LIN {X 0,Y 284.556,Z 208.031,A -85,B 0,C 180,E1 -16929.956,E2 -16929.956} C_VEL
LIN {X 0,Y 284.452,Z 208.046,A -85,B 0,C 180,E1 -16934.304,E2 -16934.304} C_VEL
LIN {X 0,Y 284.322,Z 208.068,A -85,B 0,C 180,E1 -16938.744,E2 -16938.744} C_VEL
LIN {X 0,Y 284.299,Z 208.074,A -85,B 0,C 180,E1 -16943.299,E2 -16943.299} C_VEL
LIN {X 0,Y 284.315,Z 208.073,A -85,B 0,C 180,E1 -16947.146,E2 -16947.146} C_VEL
LIN {X 0,Y 284.286,Z 208.075,A -85,B 0,C 180,E1 -16950.093,E2 -16950.093} C_VEL
LIN {X 0,Y 284.295,Z 208.073,A -85,B 0,C 180,E1 -16952.947,E2 -16952.947} C_VEL
LIN {X 0,Y 284.312,Z 208.07,A -85,B 0,C 180,E1 -16956.389,E2 -16956.389} C_VEL
LIN {X 0,Y 284.299,Z 208.15,A -85,B 0,C 180,E1 -16959.192,E2 -16959.192} C_VEL
LIN {X 0,Y 286.105,Z 215.668,A -85,B 0,C 180,E1 -16963.457,E2 -16963.457} C_VEL
LIN {X 0,Y 287.767,Z 222.743,A -85,B 0,C 180,E1 -16967.111,E2 -16967.111} C_VEL
LIN {X 0,Y 289.38,Z 229.741,A -85,B 0,C 180,E1 -16970.407,E2 -16970.407} C_VEL
LIN {X 0,Y 291.264,Z 238.5,A -85,B 0,C 180,E1 -16974.224,E2 -16974.224} C_VEL
LIN {X 0,Y 292.271,Z 243.914,A -85,B 0,C 180,E1 -16976.425,E2 -16976.425} C_VEL
LIN {X 0,Y 290.199,Z 252.267,A -85,B 0,C 180,E1 -16979.433,E2 -16979.433} C_VEL
LIN {X 0,Y 286.998,Z 266.482,A -85,B 0,C 180,E1 -16984.573,E2 -16984.573} C_VEL
LIN {X 0,Y 285.727,Z 273,A -85,B 0,C 180,E1 -16986.97,E2 -16986.97} C_VEL
LIN {X 0,Y 286.996,Z 286.111,A -85,B 0,C 180,E1 -16987.696,E2 -16987.696} C_VEL
LIN {X 0,Y 287.368,Z 299.101,A -85,B 0,C 180,E1 -16988.692,E2 -16988.692} C_VEL
LIN {X 0,Y 287.659,Z 310.186,A -85,B 0,C 180,E1 -16989.821,E2 -16989.821} C_VEL
LIN {X 0,Y 287.568,Z 320.328,A -85,B 0,C 180,E1 -16991.108,E2 -16991.108} C_VEL
LIN {X 0,Y 286.441,Z 329.749,A -85,B 0,C 180,E1 -16992.511,E2 -16992.511} C_VEL
LIN {X 0,Y 285.855,Z 335.833,A -85,B 0,C 180,E1 -16993.507,E2 -16993.507} C_VEL
LIN {X 0,Y 284.785,Z 346.52,A -85,B 0,C 180,E1 -16995.167,E2 -16995.167} C_VEL
LIN {X 0,Y 283.948,Z 356.755,A -85,B 0,C 180,E1 -16997.131,E2 -16997.131} C_VEL
LIN {X 0,Y 283.401,Z 364.415,A -85,B 0,C 180,E1 -16998.921,E2 -16998.921} C_VEL
LIN {X 0,Y 283.048,Z 371.92,A -85,B 0,C 180,E1 -17001.074,E2 -17001.074} C_VEL
LIN {X 0,Y 282.887,Z 378.816,A -85,B 0,C 180,E1 -17003.595,E2 -17003.595} C_VEL
LIN {X 0,Y 282.821,Z 383.257,A -85,B 0,C 180,E1 -17005.727,E2 -17005.727} C_VEL
LIN {X 0,Y 282.938,Z 385.581,A -85,B 0,C 180,E1 -17007.154,E2 -17007.154} C_VEL
LIN {X 0,Y 282.983,Z 387.424,A -85,B 0,C 180,E1 -17008.579,E2 -17008.579} C_VEL
LIN {X 0,Y 282.977,Z 388.816,A -85,B 0,C 180,E1 -17010.002,E2 -17010.002} C_VEL
LIN {X 0,Y 282.898,Z 389.732,A -85,B 0,C 180,E1 -17011.425,E2 -17011.425} C_VEL
LIN {X 0,Y 282.576,Z 390.303,A -85,B 0,C 180,E1 -17014.281,E2 -17014.281} C_VEL
LIN {X 0,Y 282.524,Z 389.999,A -85,B 0,C 180,E1 -17015.712,E2 -17015.712} C_VEL
LIN {X 0,Y 282.839,Z 388.158,A -85,B 0,C 180,E1 -17018.576,E2 -17018.576} C_VEL
LIN {X 0,Y 283.775,Z 384.776,A -85,B 0,C 180,E1 -17021.429,E2 -17021.429} C_VEL
LIN {X 0,Y 284.906,Z 381.163,A -85,B 0,C 180,E1 -17023.555,E2 -17023.555} C_VEL
LIN {X 0,Y 286.668,Z 376.58,A -85,B 0,C 180,E1 -17025.647,E2 -17025.647} C_VEL
LIN {X 0,Y 288.918,Z 369.965,A -85,B 0,C 180,E1 -17028.07,E2 -17028.07} C_VEL
LIN {X 0,Y 291.48,Z 363.007,A -85,B 0,C 180,E1 -17030.097,E2 -17030.097} C_VEL
LIN {X 0,Y 295.275,Z 353.149,A -85,B 0,C 180,E1 -17032.386,E2 -17032.386} C_VEL
LIN {X 0,Y 298.964,Z 342.899,A -85,B 0,C 180,E1 -17034.294,E2 -17034.294} C_VEL
LIN {X 0,Y 302.662,Z 331.714,A -85,B 0,C 180,E1 -17035.996,E2 -17035.996} C_VEL
LIN {X 0,Y 305.228,Z 321.28,A -85,B 0,C 180,E1 -17037.421,E2 -17037.421} C_VEL
LIN {X 0,Y 306.812,Z 309.853,A -85,B 0,C 180,E1 -17038.948,E2 -17038.948} C_VEL
LIN {X 0,Y 307.335,Z 299.297,A -85,B 0,C 180,E1 -17040.382,E2 -17040.382} C_VEL
LIN {X 0,Y 306.766,Z 286.625,A -85,B 0,C 180,E1 -17042.257,E2 -17042.257} C_VEL
LIN {X 0,Y 305.752,Z 277.475,A -85,B 0,C 180,E1 -17043.754,E2 -17043.754} C_VEL
LIN {X 0,Y 304.821,Z 269.242,A -85,B 0,C 180,E1 -17045.302,E2 -17045.302} C_VEL
LIN {X 0,Y 305.142,Z 266.775,A -85,B 0,C 180,E1 -17046.281,E2 -17046.281} C_VEL
LIN {X 0,Y 305.029,Z 262.987,A -85,B 0,C 180,E1 -17048.471,E2 -17048.471} C_VEL
LIN {X 0,Y 304.799,Z 260.629,A -85,B 0,C 180,E1 -17050.456,E2 -17050.456} C_VEL
LIN {X 0,Y 304.213,Z 259.405,A -85,B 0,C 180,E1 -17052.33,E2 -17052.33} C_VEL
LIN {X 0,Y 303.415,Z 259.011,A -85,B 0,C 180,E1 -17054.106,E2 -17054.106} C_VEL
LIN {X 0,Y 302.635,Z 259.068,A -85,B 0,C 180,E1 -17056.048,E2 -17056.048} C_VEL
LIN {X 0,Y 301.48,Z 260.13,A -85,B 0,C 180,E1 -17059.252,E2 -17059.252} C_VEL
LIN {X 0,Y 300.921,Z 261.159,A -85,B 0,C 180,E1 -17060.907,E2 -17060.907} C_VEL
LIN {X 0,Y 300.012,Z 262.974,A -85,B 0,C 180,E1 -17062.651,E2 -17062.651} C_VEL
LIN {X 0,Y 301.617,Z 268.449,A -85,B 0,C 180,E1 -17064.643,E2 -17064.643} C_VEL
LIN {X 0,Y 304.148,Z 276.846,A -85,B 0,C 180,E1 -17067.224,E2 -17067.224} C_VEL
LIN {X 0,Y 306.842,Z 287.914,A -85,B 0,C 180,E1 -17070.05,E2 -17070.05} C_VEL
LIN {X 0,Y 308.147,Z 297.139,A -85,B 0,C 180,E1 -17072.074,E2 -17072.074} C_VEL
LIN {X 0,Y 308.384,Z 304.136,A -85,B 0,C 180,E1 -17073.478,E2 -17073.478} C_VEL
LIN {X 0,Y 304.667,Z 315.586,A -85,B 0,C 180,E1 -17075.103,E2 -17075.103} C_VEL
LIN {X 0,Y 300.868,Z 326.03,A -85,B 0,C 180,E1 -17076.967,E2 -17076.967} C_VEL
LIN {X 0,Y 297.408,Z 334.701,A -85,B 0,C 180,E1 -17078.877,E2 -17078.877} C_VEL
LIN {X 0,Y 293.88,Z 342.88,A -85,B 0,C 180,E1 -17081.165,E2 -17081.165} C_VEL
LIN {X 0,Y 291.288,Z 348.565,A -85,B 0,C 180,E1 -17083.17,E2 -17083.17} C_VEL
LIN {X 0,Y 289.185,Z 353.139,A -85,B 0,C 180,E1 -17085.216,E2 -17085.216} C_VEL
LIN {X 0,Y 287.297,Z 356.739,A -85,B 0,C 180,E1 -17087.281,E2 -17087.281} C_VEL
LIN {X 0,Y 285.522,Z 359.952,A -85,B 0,C 180,E1 -17089.933,E2 -17089.933} C_VEL
LIN {X 0,Y 284.505,Z 361.163,A -85,B 0,C 180,E1 -17091.477,E2 -17091.477} C_VEL
LIN {X 0,Y 283.599,Z 362.166,A -85,B 0,C 180,E1 -17094.311,E2 -17094.311} C_VEL
LIN {X 0,Y 283.258,Z 362.063,A -85,B 0,C 180,E1 -17095.731,E2 -17095.731} C_VEL
LIN {X 0,Y 282.702,Z 360.712,A -85,B 0,C 180,E1 -17098.576,E2 -17098.576} C_VEL
LIN {X 0,Y 282.565,Z 359.447,A -85,B 0,C 180,E1 -17100,E2 -17100} C_VEL
LIN {X 0,Y 282.563,Z 356.745,A -85,B 0,C 180,E1 -17102.138,E2 -17102.138} C_VEL
LIN {X 0,Y 282.716,Z 353.044,A -85,B 0,C 180,E1 -17104.277,E2 -17104.277} C_VEL
LIN {X 0,Y 282.917,Z 347.475,A -85,B 0,C 180,E1 -17106.712,E2 -17106.712} C_VEL
LIN {X 0,Y 283.339,Z 341.061,A -85,B 0,C 180,E1 -17108.918,E2 -17108.918} C_VEL
LIN {X 0,Y 283.988,Z 333.386,A -85,B 0,C 180,E1 -17111.058,E2 -17111.058} C_VEL
LIN {X 0,Y 284.831,Z 323.888,A -85,B 0,C 180,E1 -17113.193,E2 -17113.193} C_VEL
LIN {X 0,Y 285.828,Z 314.315,A -85,B 0,C 180,E1 -17114.962,E2 -17114.962} C_VEL
LIN {X 0,Y 286.847,Z 302.522,A -85,B 0,C 180,E1 -17116.732,E2 -17116.732} C_VEL
LIN {X 0,Y 287.821,Z 291.265,A -85,B 0,C 180,E1 -17118.103,E2 -17118.103} C_VEL
LIN {X 0,Y 288.584,Z 280.158,A -85,B 0,C 180,E1 -17119.194,E2 -17119.194} C_VEL
LIN {X 0,Y 286.473,Z 266.68,A -85,B 0,C 180,E1 -17120.318,E2 -17120.318} C_VEL
LIN {X 0,Y 284.567,Z 252.884,A -85,B 0,C 180,E1 -17121.173,E2 -17121.173} C_VEL
LIN {X 0,Y 284.521,Z 252.298,A -85,B 0,C 180,E1 -17121.24,E2 -17121.24} C_VEL
LIN {X 0,Y 284.94,Z 244.617,A -85,B 0,C 180,E1 -17124.791,E2 -17124.791} C_VEL
LIN {X 0,Y 285.368,Z 236.232,A -85,B 0,C 180,E1 -17128.702,E2 -17128.702} C_VEL
LIN {X 0,Y 285.937,Z 227.639,A -85,B 0,C 180,E1 -17132.734,E2 -17132.734} C_VEL
LIN {X 0,Y 286.29,Z 220.567,A -85,B 0,C 180,E1 -17136.098,E2 -17136.098} C_VEL
LIN {X 0,Y 285.648,Z 214.901,A -85,B 0,C 180,E1 -17138.886,E2 -17138.886} C_VEL
LIN {X 0,Y 284.363,Z 208.065,A -85,B 0,C 180,E1 -17142.352,E2 -17142.352} C_VEL
LIN {X 0,Y 284.262,Z 208.078,A -85,B 0,C 180,E1 -17146.188,E2 -17146.188} C_VEL
LIN {X 0,Y 284.312,Z 208.072,A -85,B 0,C 180,E1 -17150.023,E2 -17150.023} C_VEL
LIN {X 0,Y 284.326,Z 208.072,A -85,B 0,C 180,E1 -17153.611,E2 -17153.611} C_VEL
LIN {X 0,Y 284.368,Z 208.282,A -85,B 0,C 180,E1 -17155.007,E2 -17155.007} C_VEL
LIN {X 0,Y 284.692,Z 210.194,A -85,B 0,C 180,E1 -17157.103,E2 -17157.103} C_VEL
LIN {X 0,Y 284.913,Z 213.447,A -85,B 0,C 180,E1 -17160.438,E2 -17160.438} C_VEL
LIN {X 0,Y 284.838,Z 216.778,A -85,B 0,C 180,E1 -17163.631,E2 -17163.631} C_VEL
LIN {X 0,Y 284.709,Z 220.161,A -85,B 0,C 180,E1 -17166.735,E2 -17166.735} C_VEL
LIN {X 0,Y 284.654,Z 223.645,A -85,B 0,C 180,E1 -17169.776,E2 -17169.776} C_VEL
LIN {X 0,Y 284.578,Z 226.72,A -85,B 0,C 180,E1 -17172.321,E2 -17172.321} C_VEL
LIN {X 0,Y 287.73,Z 237.495,A -85,B 0,C 180,E1 -17173.172,E2 -17173.172} C_VEL
LIN {X 0,Y 290.174,Z 247.752,A -85,B 0,C 180,E1 -17174.248,E2 -17174.248} C_VEL
LIN {X 0,Y 291.01,Z 253.902,A -85,B 0,C 180,E1 -17175.021,E2 -17175.021} C_VEL
LIN {X 0,Y 290.089,Z 263.238,A -85,B 0,C 180,E1 -17176.335,E2 -17176.335} C_VEL
LIN {X 0,Y 289.359,Z 269.037,A -85,B 0,C 180,E1 -17177.372,E2 -17177.372} C_VEL
LIN {X 0,Y 288.305,Z 275.346,A -85,B 0,C 180,E1 -17178.753,E2 -17178.753} C_VEL
LIN {X 0,Y 287.394,Z 280.335,A -85,B 0,C 180,E1 -17180.142,E2 -17180.142} C_VEL
LIN {X 0,Y 286.592,Z 284.326,A -85,B 0,C 180,E1 -17181.537,E2 -17181.537} C_VEL
LIN {X 0,Y 286.092,Z 288.746,A -85,B 0,C 180,E1 -17183.652,E2 -17183.652} C_VEL
LIN {X 0,Y 285.241,Z 291.75,A -85,B 0,C 180,E1 -17185.759,E2 -17185.759} C_VEL
LIN {X 0,Y 285.065,Z 293.009,A -85,B 0,C 180,E1 -17187.172,E2 -17187.172} C_VEL
LIN {X 0,Y 284.86,Z 293.775,A -85,B 0,C 180,E1 -17188.584,E2 -17188.584} C_VEL
LIN {X 0,Y 284.777,Z 294.043,A -85,B 0,C 180,E1 -17189.998,E2 -17189.998} C_VEL
LIN {X 0,Y 284.858,Z 293.811,A -85,B 0,C 180,E1 -17191.412,E2 -17191.412} C_VEL
LIN {X 0,Y 285.061,Z 293.095,A -85,B 0,C 180,E1 -17192.824,E2 -17192.824} C_VEL
LIN {X 0,Y 285.238,Z 291.887,A -85,B 0,C 180,E1 -17194.237,E2 -17194.237} C_VEL
LIN {X 0,Y 286.082,Z 288.958,A -85,B 0,C 180,E1 -17196.345,E2 -17196.345} C_VEL
LIN {X 0,Y 286.554,Z 284.623,A -85,B 0,C 180,E1 -17198.46,E2 -17198.46} C_VEL
LIN {X 0,Y 287.252,Z 281.745,A -85,B 0,C 180,E1 -17199.504,E2 -17199.504} C_VEL
LIN {X 0,Y 288.046,Z 277.103,A -85,B 0,C 180,E1 -17200.898,E2 -17200.898} C_VEL
LIN {X 0,Y 289.079,Z 271.275,A -85,B 0,C 180,E1 -17202.28,E2 -17202.28} C_VEL
LIN {X 0,Y 289.917,Z 264.953,A -85,B 0,C 180,E1 -17203.491,E2 -17203.491} C_VEL
LIN {X 0,Y 290.611,Z 257.713,A -85,B 0,C 180,E1 -17204.606,E2 -17204.606} C_VEL
LIN {X 0,Y 291.046,Z 252.834,A -85,B 0,C 180,E1 -17205.231,E2 -17205.231} C_VEL
LIN {X 0,Y 289.66,Z 245.069,A -85,B 0,C 180,E1 -17206.177,E2 -17206.177} C_VEL
LIN {X 0,Y 286.946,Z 234.411,A -85,B 0,C 180,E1 -17207.213,E2 -17207.213} C_VEL
LIN {X 0,Y 284.582,Z 226.689,A -85,B 0,C 180,E1 -17207.839,E2 -17207.839} C_VEL
LIN {X 0,Y 284.672,Z 223.765,A -85,B 0,C 180,E1 -17210.256,E2 -17210.256} C_VEL
LIN {X 0,Y 284.791,Z 218.619,A -85,B 0,C 180,E1 -17214.802,E2 -17214.802} C_VEL
LIN {X 0,Y 284.886,Z 215.255,A -85,B 0,C 180,E1 -17217.949,E2 -17217.949} C_VEL
LIN {X 0,Y 284.815,Z 211.982,A -85,B 0,C 180,E1 -17221.208,E2 -17221.208} C_VEL
LIN {X 0,Y 284.444,Z 208.769,A -85,B 0,C 180,E1 -17224.628,E2 -17224.628} C_VEL
LIN {X 0,Y 284.344,Z 208.067,A -85,B 0,C 180,E1 -17225.512,E2 -17225.512} C_VEL
LIN {X 0,Y 284.318,Z 208.069,A -85,B 0,C 180,E1 -17228.165,E2 -17228.165} C_VEL
LIN {X 0,Y 284.263,Z 208.075,A -85,B 0,C 180,E1 -17232.123,E2 -17232.123} C_VEL
LIN {X 0,Y 284.279,Z 208.071,A -85,B 0,C 180,E1 -17236.193,E2 -17236.193} C_VEL
LIN {X 0,Y 284.305,Z 208.067,A -85,B 0,C 180,E1 -17240.021,E2 -17240.021} C_VEL
LIN {X 0,Y 284.326,Z 208.066,A -85,B 0,C 180,E1 -17243.613,E2 -17243.613} C_VEL
LIN {X 0,Y 284.301,Z 208.067,A -85,B 0,C 180,E1 -17247.188,E2 -17247.188} C_VEL
LIN {X 0,Y 284.351,Z 208.056,A -85,B 0,C 180,E1 -17250.375,E2 -17250.375} C_VEL
LIN {X 0,Y 284.369,Z 208.061,A -85,B 0,C 180,E1 -17253.585,E2 -17253.585} C_VEL
LIN {X 0,Y 284.357,Z 208.064,A -85,B 0,C 180,E1 -17256.706,E2 -17256.706} C_VEL
LIN {X 0,Y 284.394,Z 208.056,A -85,B 0,C 180,E1 -17261.261,E2 -17261.261} C_VEL
LIN {X 0,Y 284.482,Z 208.035,A -85,B 0,C 180,E1 -17264.458,E2 -17264.458} C_VEL
LIN {X 0,Y 284.477,Z 208.046,A -85,B 0,C 180,E1 -17268.601,E2 -17268.601} C_VEL
LIN {X 0,Y 284.628,Z 208.024,A -85,B 0,C 180,E1 -17271.48,E2 -17271.48} C_VEL
LIN {X 0,Y 284.586,Z 208.026,A -85,B 0,C 180,E1 -17274.331,E2 -17274.331} C_VEL
LIN {X 0,Y 284.844,Z 207.997,A -85,B 0,C 180,E1 -17278.76,E2 -17278.76} C_VEL
LIN {X 0,Y 284.138,Z 208.08,A -85,B 0,C 180,E1 -17279.941,E2 -17279.941} C_VEL
LIN {X 0,Y 281.114,Z 208.466,A -85,B 0,C 180,E1 -17281.859,E2 -17281.859} C_VEL
LIN {X 0,Y 278.579,Z 208.78,A -85,B 0,C 180,E1 -17283.418,E2 -17283.418} C_VEL
LIN {X 0,Y 277.537,Z 208.903,A -85,B 0,C 180,E1 -17284.63,E2 -17284.63} C_VEL
LIN {X 0,Y 277.478,Z 208.911,A -85,B 0,C 180,E1 -17285.041,E2 -17285.041} C_VEL
LIN {X 0,Y 277.642,Z 208.9,A -85,B 0,C 180,E1 -17287.271,E2 -17287.271} C_VEL
LIN {X 0,Y 277.496,Z 208.912,A -85,B 0,C 180,E1 -17290.212,E2 -17290.212} C_VEL
LIN {X 0,Y 277.398,Z 208.928,A -85,B 0,C 180,E1 -17294.676,E2 -17294.676} C_VEL
LIN {X 0,Y 277.274,Z 208.948,A -85,B 0,C 180,E1 -17299.239,E2 -17299.239} C_VEL
LIN {X 0,Y 277.249,Z 208.952,A -85,B 0,C 180,E1 -17303.928,E2 -17303.928} C_VEL
LIN {X 0,Y 277.256,Z 208.951,A -85,B 0,C 180,E1 -17307.482,E2 -17307.482} C_VEL
LIN {X 0,Y 277.238,Z 208.952,A -85,B 0,C 180,E1 -17310.474,E2 -17310.474} C_VEL
LIN {X 0,Y 277.236,Z 208.947,A -85,B 0,C 180,E1 -17313.897,E2 -17313.897} C_VEL
LIN {X 0,Y 277.263,Z 208.948,A -85,B 0,C 180,E1 -17317.845,E2 -17317.845} C_VEL
LIN {X 0,Y 277.289,Z 209.153,A -85,B 0,C 180,E1 -17318.218,E2 -17318.218} C_VEL
LIN {X 0,Y 278.743,Z 215.264,A -85,B 0,C 180,E1 -17321.925,E2 -17321.925} C_VEL
LIN {X 0,Y 280.48,Z 222.527,A -85,B 0,C 180,E1 -17325.832,E2 -17325.832} C_VEL
LIN {X 0,Y 282.263,Z 230.179,A -85,B 0,C 180,E1 -17329.659,E2 -17329.659} C_VEL
LIN {X 0,Y 284.092,Z 238.844,A -85,B 0,C 180,E1 -17333.581,E2 -17333.581} C_VEL
LIN {X 0,Y 285.287,Z 245.368,A -85,B 0,C 180,E1 -17336.342,E2 -17336.342} C_VEL
LIN {X 0,Y 282.547,Z 255.692,A -85,B 0,C 180,E1 -17340.169,E2 -17340.169} C_VEL
LIN {X 0,Y 279.795,Z 267.845,A -85,B 0,C 180,E1 -17344.724,E2 -17344.724} C_VEL
LIN {X 0,Y 278.89,Z 272.292,A -85,B 0,C 180,E1 -17346.421,E2 -17346.421} C_VEL
LIN {X 0,Y 280.198,Z 286.506,A -85,B 0,C 180,E1 -17347.27,E2 -17347.27} C_VEL
LIN {X 0,Y 280.535,Z 297.591,A -85,B 0,C 180,E1 -17348.147,E2 -17348.147} C_VEL
LIN {X 0,Y 280.705,Z 309.027,A -85,B 0,C 180,E1 -17349.319,E2 -17349.319} C_VEL
LIN {X 0,Y 280.696,Z 319.136,A -85,B 0,C 180,E1 -17350.627,E2 -17350.627} C_VEL
LIN {X 0,Y 279.807,Z 327.565,A -85,B 0,C 180,E1 -17351.893,E2 -17351.893} C_VEL
LIN {X 0,Y 278.362,Z 339.738,A -85,B 0,C 180,E1 -17354.066,E2 -17354.066} C_VEL
LIN {X 0,Y 277.479,Z 349.307,A -85,B 0,C 180,E1 -17355.705,E2 -17355.705} C_VEL
LIN {X 0,Y 276.636,Z 359.657,A -85,B 0,C 180,E1 -17357.904,E2 -17357.904} C_VEL
LIN {X 0,Y 276.09,Z 368.004,A -85,B 0,C 180,E1 -17360.108,E2 -17360.108} C_VEL
LIN {X 0,Y 275.934,Z 373.705,A -85,B 0,C 180,E1 -17361.949,E2 -17361.949} C_VEL
LIN {X 0,Y 275.856,Z 379.204,A -85,B 0,C 180,E1 -17364.153,E2 -17364.153} C_VEL
LIN {X 0,Y 275.829,Z 383.434,A -85,B 0,C 180,E1 -17366.35,E2 -17366.35} C_VEL
LIN {X 0,Y 275.93,Z 386.546,A -85,B 0,C 180,E1 -17368.542,E2 -17368.542} C_VEL
LIN {X 0,Y 275.922,Z 388.02,A -85,B 0,C 180,E1 -17370.002,E2 -17370.002} C_VEL
LIN {X 0,Y 275.833,Z 389.057,A -85,B 0,C 180,E1 -17371.462,E2 -17371.462} C_VEL
LIN {X 0,Y 275.515,Z 389.644,A -85,B 0,C 180,E1 -17372.926,E2 -17372.926} C_VEL
LIN {X 0,Y 275.453,Z 389.649,A -85,B 0,C 180,E1 -17375.696,E2 -17375.696} C_VEL
LIN {X 0,Y 275.526,Z 389.004,A -85,B 0,C 180,E1 -17377.329,E2 -17377.329} C_VEL
LIN {X 0,Y 275.797,Z 388.026,A -85,B 0,C 180,E1 -17378.797,E2 -17378.797} C_VEL
LIN {X 0,Y 276.795,Z 384.854,A -85,B 0,C 180,E1 -17381.722,E2 -17381.722} C_VEL
LIN {X 0,Y 277.992,Z 381.459,A -85,B 0,C 180,E1 -17383.898,E2 -17383.898} C_VEL
LIN {X 0,Y 280.551,Z 375.462,A -85,B 0,C 180,E1 -17386.745,E2 -17386.745} C_VEL
LIN {X 0,Y 283.08,Z 368.624,A -85,B 0,C 180,E1 -17389.244,E2 -17389.244} C_VEL
LIN {X 0,Y 286.534,Z 360.394,A -85,B 0,C 180,E1 -17391.589,E2 -17391.589} C_VEL
LIN {X 0,Y 290.099,Z 351.783,A -85,B 0,C 180,E1 -17393.563,E2 -17393.563} C_VEL
LIN {X 0,Y 294.129,Z 341.451,A -85,B 0,C 180,E1 -17395.475,E2 -17395.475} C_VEL
LIN {X 0,Y 297.935,Z 330.338,A -85,B 0,C 180,E1 -17397.198,E2 -17397.198} C_VEL
LIN {X 0,Y 300.617,Z 319.331,A -85,B 0,C 180,E1 -17398.76,E2 -17398.76} C_VEL
LIN {X 0,Y 302.234,Z 307.982,A -85,B 0,C 180,E1 -17400.358,E2 -17400.358} C_VEL
LIN {X 0,Y 302.693,Z 296.454,A -85,B 0,C 180,E1 -17402.099,E2 -17402.099} C_VEL
LIN {X 0,Y 302.356,Z 285.308,A -85,B 0,C 180,E1 -17403.91,E2 -17403.91} C_VEL
LIN {X 0,Y 301.381,Z 274.903,A -85,B 0,C 180,E1 -17405.87,E2 -17405.87} C_VEL
LIN {X 0,Y 300.858,Z 272.433,A -85,B 0,C 180,E1 -17406.511,E2 -17406.511} C_VEL
LIN {X 0,Y 299.528,Z 268.255,A -85,B 0,C 180,E1 -17408.065,E2 -17408.065} C_VEL
LIN {X 0,Y 299.467,Z 266.402,A -85,B 0,C 180,E1 -17409.321,E2 -17409.321} C_VEL
LIN {X 0,Y 299.006,Z 264.514,A -85,B 0,C 180,E1 -17411.223,E2 -17411.223} C_VEL
LIN {X 0,Y 298.23,Z 263.565,A -85,B 0,C 180,E1 -17413.112,E2 -17413.112} C_VEL
LIN {X 0,Y 297.267,Z 263.279,A -85,B 0,C 180,E1 -17415.177,E2 -17415.177} C_VEL
LIN {X 0,Y 295.998,Z 263.852,A -85,B 0,C 180,E1 -17418.332,E2 -17418.332} C_VEL
LIN {X 0,Y 295.723,Z 264.277,A -85,B 0,C 180,E1 -17419.189,E2 -17419.189} C_VEL
LIN {X 0,Y 297.195,Z 268.792,A -85,B 0,C 180,E1 -17422.059,E2 -17422.059} C_VEL
LIN {X 0,Y 298.351,Z 273.545,A -85,B 0,C 180,E1 -17423.921,E2 -17423.921} C_VEL
LIN {X 0,Y 300.127,Z 281.201,A -85,B 0,C 180,E1 -17426.42,E2 -17426.42} C_VEL
LIN {X 0,Y 302.144,Z 291.405,A -85,B 0,C 180,E1 -17429.221,E2 -17429.221} C_VEL
LIN {X 0,Y 303.018,Z 299.258,A -85,B 0,C 180,E1 -17431.089,E2 -17431.089} C_VEL
LIN {X 0,Y 303.194,Z 305.086,A -85,B 0,C 180,E1 -17432.38,E2 -17432.38} C_VEL
LIN {X 0,Y 303.03,Z 306.944,A -85,B 0,C 180,E1 -17432.745,E2 -17432.745} C_VEL
LIN {X 0,Y 299.389,Z 317.16,A -85,B 0,C 180,E1 -17434.261,E2 -17434.261} C_VEL
LIN {X 0,Y 295.34,Z 327.36,A -85,B 0,C 180,E1 -17436.138,E2 -17436.138} C_VEL
LIN {X 0,Y 291.691,Z 335.803,A -85,B 0,C 180,E1 -17438.071,E2 -17438.071} C_VEL
LIN {X 0,Y 287.904,Z 343.832,A -85,B 0,C 180,E1 -17440.388,E2 -17440.388} C_VEL
LIN {X 0,Y 284.688,Z 350.235,A -85,B 0,C 180,E1 -17442.768,E2 -17442.768} C_VEL
LIN {X 0,Y 282.463,Z 354.544,A -85,B 0,C 180,E1 -17444.856,E2 -17444.856} C_VEL
LIN {X 0,Y 280.498,Z 357.916,A -85,B 0,C 180,E1 -17446.968,E2 -17446.968} C_VEL
LIN {X 0,Y 278.517,Z 360.953,A -85,B 0,C 180,E1 -17449.826,E2 -17449.826} C_VEL
LIN {X 0,Y 277.528,Z 361.939,A -85,B 0,C 180,E1 -17451.261,E2 -17451.261} C_VEL
LIN {X 0,Y 276.917,Z 362.505,A -85,B 0,C 180,E1 -17452.71,E2 -17452.71} C_VEL
LIN {X 0,Y 276.548,Z 362.662,A -85,B 0,C 180,E1 -17454.166,E2 -17454.166} C_VEL
LIN {X 0,Y 276.191,Z 362.455,A -85,B 0,C 180,E1 -17455.622,E2 -17455.622} C_VEL
LIN {X 0,Y 275.842,Z 361.877,A -85,B 0,C 180,E1 -17457.079,E2 -17457.079} C_VEL
LIN {X 0,Y 275.616,Z 360.891,A -85,B 0,C 180,E1 -17458.539,E2 -17458.539} C_VEL
LIN {X 0,Y 275.466,Z 357.675,A -85,B 0,C 180,E1 -17461.462,E2 -17461.462} C_VEL
LIN {X 0,Y 275.601,Z 354.143,A -85,B 0,C 180,E1 -17463.655,E2 -17463.655} C_VEL
LIN {X 0,Y 275.724,Z 348.651,A -85,B 0,C 180,E1 -17466.224,E2 -17466.224} C_VEL
LIN {X 0,Y 276.218,Z 341.497,A -85,B 0,C 180,E1 -17468.781,E2 -17468.781} C_VEL
LIN {X 0,Y 276.845,Z 333.843,A -85,B 0,C 180,E1 -17470.976,E2 -17470.976} C_VEL
LIN {X 0,Y 277.684,Z 324.356,A -85,B 0,C 180,E1 -17473.167,E2 -17473.167} C_VEL
LIN {X 0,Y 278.794,Z 313.745,A -85,B 0,C 180,E1 -17475.162,E2 -17475.162} C_VEL
LIN {X 0,Y 279.753,Z 303.135,A -85,B 0,C 180,E1 -17476.788,E2 -17476.788} C_VEL
LIN {X 0,Y 280.755,Z 291.635,A -85,B 0,C 180,E1 -17478.234,E2 -17478.234} C_VEL
LIN {X 0,Y 281.534,Z 281.007,A -85,B 0,C 180,E1 -17479.315,E2 -17479.315} C_VEL
LIN {X 0,Y 279.378,Z 266.893,A -85,B 0,C 180,E1 -17480.525,E2 -17480.525} C_VEL
LIN {X 0,Y 277.475,Z 252.691,A -85,B 0,C 180,E1 -17481.439,E2 -17481.439} C_VEL
LIN {X 0,Y 277.966,Z 244.118,A -85,B 0,C 180,E1 -17485.457,E2 -17485.457} C_VEL
LIN {X 0,Y 278.417,Z 235.601,A -85,B 0,C 180,E1 -17489.488,E2 -17489.488} C_VEL
LIN {X 0,Y 278.932,Z 228.638,A -85,B 0,C 180,E1 -17492.801,E2 -17492.801} C_VEL
LIN {X 0,Y 279.27,Z 222.266,A -85,B 0,C 180,E1 -17495.859,E2 -17495.859} C_VEL
LIN {X 0,Y 278.964,Z 218.209,A -85,B 0,C 180,E1 -17497.876,E2 -17497.876} C_VEL
LIN {X 0,Y 277.632,Z 210.663,A -85,B 0,C 180,E1 -17501.687,E2 -17501.687} C_VEL
LIN {X 0,Y 277.304,Z 208.945,A -85,B 0,C 180,E1 -17502.626,E2 -17502.626} C_VEL
LIN {X 0,Y 277.221,Z 208.952,A -85,B 0,C 180,E1 -17507.324,E2 -17507.324} C_VEL
LIN {X 0,Y 277.262,Z 208.953,A -85,B 0,C 180,E1 -17511.794,E2 -17511.794} C_VEL
LIN {X 0,Y 277.305,Z 209.052,A -85,B 0,C 180,E1 -17514.195,E2 -17514.195} C_VEL
LIN {X 0,Y 277.805,Z 212.464,A -85,B 0,C 180,E1 -17517.907,E2 -17517.907} C_VEL
LIN {X 0,Y 277.931,Z 215.745,A -85,B 0,C 180,E1 -17521.283,E2 -17521.283} C_VEL
LIN {X 0,Y 277.823,Z 220.273,A -85,B 0,C 180,E1 -17525.6,E2 -17525.6} C_VEL
LIN {X 0,Y 277.672,Z 224.609,A -85,B 0,C 180,E1 -17529.47,E2 -17529.47} C_VEL
LIN {X 0,Y 277.613,Z 227.461,A -85,B 0,C 180,E1 -17531.793,E2 -17531.793} C_VEL
LIN {X 0,Y 280.661,Z 237.687,A -85,B 0,C 180,E1 -17532.625,E2 -17532.625} C_VEL
LIN {X 0,Y 283.139,Z 247.63,A -85,B 0,C 180,E1 -17533.689,E2 -17533.689} C_VEL
LIN {X 0,Y 284.219,Z 255.206,A -85,B 0,C 180,E1 -17534.66,E2 -17534.66} C_VEL
LIN {X 0,Y 283.283,Z 264.343,A -85,B 0,C 180,E1 -17536,E2 -17536} C_VEL
LIN {X 0,Y 282.522,Z 270.096,A -85,B 0,C 180,E1 -17537.061,E2 -17537.061} C_VEL
LIN {X 0,Y 281.424,Z 276.38,A -85,B 0,C 180,E1 -17538.474,E2 -17538.474} C_VEL
LIN {X 0,Y 280.473,Z 281.342,A -85,B 0,C 180,E1 -17539.896,E2 -17539.896} C_VEL
LIN {X 0,Y 279.641,Z 285.319,A -85,B 0,C 180,E1 -17541.325,E2 -17541.325} C_VEL
LIN {X 0,Y 279.108,Z 289.729,A -85,B 0,C 180,E1 -17543.492,E2 -17543.492} C_VEL
LIN {X 0,Y 278.234,Z 292.727,A -85,B 0,C 180,E1 -17545.652,E2 -17545.652} C_VEL
LIN {X 0,Y 278.046,Z 293.984,A -85,B 0,C 180,E1 -17547.1,E2 -17547.1} C_VEL
LIN {X 0,Y 277.835,Z 294.749,A -85,B 0,C 180,E1 -17548.549,E2 -17548.549} C_VEL
LIN {X 0,Y 277.75,Z 295.017,A -85,B 0,C 180,E1 -17549.998,E2 -17549.998} C_VEL
LIN {X 0,Y 277.833,Z 294.784,A -85,B 0,C 180,E1 -17551.448,E2 -17551.448} C_VEL
LIN {X 0,Y 278.043,Z 294.068,A -85,B 0,C 180,E1 -17552.896,E2 -17552.896} C_VEL
LIN {X 0,Y 278.231,Z 292.862,A -85,B 0,C 180,E1 -17554.344,E2 -17554.344} C_VEL
LIN {X 0,Y 279.098,Z 289.935,A -85,B 0,C 180,E1 -17556.505,E2 -17556.505} C_VEL
LIN {X 0,Y 279.603,Z 285.609,A -85,B 0,C 180,E1 -17558.672,E2 -17558.672} C_VEL
LIN {X 0,Y 280.322,Z 282.745,A -85,B 0,C 180,E1 -17559.741,E2 -17559.741} C_VEL
LIN {X 0,Y 281.148,Z 278.129,A -85,B 0,C 180,E1 -17561.169,E2 -17561.169} C_VEL
LIN {X 0,Y 282.228,Z 272.329,A -85,B 0,C 180,E1 -17562.583,E2 -17562.583} C_VEL
LIN {X 0,Y 283.109,Z 266.05,A -85,B 0,C 180,E1 -17563.822,E2 -17563.822} C_VEL
LIN {X 0,Y 283.832,Z 258.789,A -85,B 0,C 180,E1 -17564.976,E2 -17564.976} C_VEL
LIN {X 0,Y 284.247,Z 254.012,A -85,B 0,C 180,E1 -17565.612,E2 -17565.612} C_VEL
LIN {X 0,Y 282.588,Z 244.937,A -85,B 0,C 180,E1 -17566.745,E2 -17566.745} C_VEL
LIN {X 0,Y 279.806,Z 234.363,A -85,B 0,C 180,E1 -17567.79,E2 -17567.79} C_VEL
LIN {X 0,Y 277.624,Z 227.362,A -85,B 0,C 180,E1 -17568.349,E2 -17568.349} C_VEL
LIN {X 0,Y 277.689,Z 222.743,A -85,B 0,C 180,E1 -17572.309,E2 -17572.309} C_VEL
LIN {X 0,Y 277.823,Z 219.272,A -85,B 0,C 180,E1 -17575.468,E2 -17575.468} C_VEL
LIN {X 0,Y 277.932,Z 215.916,A -85,B 0,C 180,E1 -17578.712,E2 -17578.712} C_VEL
LIN {X 0,Y 277.911,Z 213.917,A -85,B 0,C 180,E1 -17580.704,E2 -17580.704} C_VEL
LIN {X 0,Y 277.589,Z 210.965,A -85,B 0,C 180,E1 -17583.846,E2 -17583.846} C_VEL
LIN {X 0,Y 277.294,Z 208.945,A -85,B 0,C 180,E1 -17586.12,E2 -17586.12} C_VEL
LIN {X 0,Y 277.233,Z 208.952,A -85,B 0,C 180,E1 -17589.325,E2 -17589.325} C_VEL
LIN {X 0,Y 277.21,Z 208.954,A -85,B 0,C 180,E1 -17593.195,E2 -17593.195} C_VEL
LIN {X 0,Y 277.231,Z 208.951,A -85,B 0,C 180,E1 -17597.318,E2 -17597.318} C_VEL
LIN {X 0,Y 277.263,Z 208.946,A -85,B 0,C 180,E1 -17601.789,E2 -17601.789} C_VEL
LIN {X 0,Y 277.277,Z 208.947,A -85,B 0,C 180,E1 -17604.34,E2 -17604.34} C_VEL
LIN {X 0,Y 277.238,Z 208.95,A -85,B 0,C 180,E1 -17607.835,E2 -17607.835} C_VEL
LIN {X 0,Y 277.281,Z 208.939,A -85,B 0,C 180,E1 -17611.211,E2 -17611.211} C_VEL
LIN {X 0,Y 277.304,Z 208.932,A -85,B 0,C 180,E1 -17614.478,E2 -17614.478} C_VEL
LIN {X 0,Y 277.276,Z 208.948,A -85,B 0,C 180,E1 -17617.654,E2 -17617.654} C_VEL
LIN {X 0,Y 277.335,Z 208.932,A -85,B 0,C 180,E1 -17620.765,E2 -17620.765} C_VEL
LIN {X 0,Y 277.424,Z 208.914,A -85,B 0,C 180,E1 -17625.325,E2 -17625.325} C_VEL
LIN {X 0,Y 277.451,Z 208.91,A -85,B 0,C 180,E1 -17629.787,E2 -17629.787} C_VEL
LIN {X 0,Y 277.63,Z 208.901,A -85,B 0,C 180,E1 -17632.728,E2 -17632.728} C_VEL
LIN {X 0,Y 277.811,Z 208.876,A -85,B 0,C 180,E1 -17638.55,E2 -17638.55} C_VEL
LIN {X 0,Y 277.81,Z 208.875,A -85,B 0,C 180,E1 -17641.45,E2 -17641.45} C_VEL
LIN {X 0,Y 277.478,Z 208.911,A -85,B 0,C 180,E1 -17645.041,E2 -17645.041} C_VEL
LIN {X 0,Y 276.87,Z 208.995,A -85,B 0,C 180,E1 -17646.255,E2 -17646.255} C_VEL
LIN {X 0,Y 274.005,Z 209.349,A -85,B 0,C 180,E1 -17648.231,E2 -17648.231} C_VEL
LIN {X 0,Y 271.532,Z 209.654,A -85,B 0,C 180,E1 -17649.838,E2 -17649.838} C_VEL
LIN {X 0,Y 270.466,Z 209.795,A -85,B 0,C 180,E1 -17651.085,E2 -17651.085} C_VEL
LIN {X 0,Y 270.379,Z 209.801,A -85,B 0,C 180,E1 -17651.507,E2 -17651.507} C_VEL
LIN {X 0,Y 270.321,Z 209.815,A -85,B 0,C 180,E1 -17655.865,E2 -17655.865} C_VEL
LIN {X 0,Y 270.231,Z 209.825,A -85,B 0,C 180,E1 -17660.574,E2 -17660.574} C_VEL
LIN {X 0,Y 270.169,Z 209.834,A -85,B 0,C 180,E1 -17664.596,E2 -17664.596} C_VEL
LIN {X 0,Y 270.186,Z 209.831,A -85,B 0,C 180,E1 -17667.918,E2 -17667.918} C_VEL
LIN {X 0,Y 270.164,Z 209.834,A -85,B 0,C 180,E1 -17671.351,E2 -17671.351} C_VEL
LIN {X 0,Y 270.189,Z 209.824,A -85,B 0,C 180,E1 -17674.907,E2 -17674.907} C_VEL
LIN {X 0,Y 270.228,Z 209.958,A -85,B 0,C 180,E1 -17677.089,E2 -17677.089} C_VEL
LIN {X 0,Y 271.454,Z 215.038,A -85,B 0,C 180,E1 -17680.335,E2 -17680.335} C_VEL
LIN {X 0,Y 272.942,Z 221.398,A -85,B 0,C 180,E1 -17684.045,E2 -17684.045} C_VEL
LIN {X 0,Y 274.874,Z 229.529,A -85,B 0,C 180,E1 -17688.338,E2 -17688.338} C_VEL
LIN {X 0,Y 276.493,Z 237.196,A -85,B 0,C 180,E1 -17691.996,E2 -17691.996} C_VEL
LIN {X 0,Y 278.254,Z 245.723,A -85,B 0,C 180,E1 -17695.81,E2 -17695.81} C_VEL
LIN {X 0,Y 278.098,Z 247.457,A -85,B 0,C 180,E1 -17696.508,E2 -17696.508} C_VEL
LIN {X 0,Y 274.677,Z 260.045,A -85,B 0,C 180,E1 -17701.334,E2 -17701.334} C_VEL
LIN {X 0,Y 272.028,Z 271.991,A -85,B 0,C 180,E1 -17705.915,E2 -17705.915} C_VEL
LIN {X 0,Y 273.269,Z 284.7,A -85,B 0,C 180,E1 -17706.66,E2 -17706.66} C_VEL
LIN {X 0,Y 273.661,Z 296.395,A -85,B 0,C 180,E1 -17707.598,E2 -17707.598} C_VEL
LIN {X 0,Y 273.753,Z 307.869,A -85,B 0,C 180,E1 -17708.79,E2 -17708.79} C_VEL
LIN {X 0,Y 273.772,Z 317.932,A -85,B 0,C 180,E1 -17710.117,E2 -17710.117} C_VEL
LIN {X 0,Y 273.181,Z 325.341,A -85,B 0,C 180,E1 -17711.244,E2 -17711.244} C_VEL
LIN {X 0,Y 271.815,Z 335.269,A -85,B 0,C 180,E1 -17713.071,E2 -17713.071} C_VEL
LIN {X 0,Y 271.056,Z 341.688,A -85,B 0,C 180,E1 -17714.397,E2 -17714.397} C_VEL
LIN {X 0,Y 270.071,Z 352.655,A -85,B 0,C 180,E1 -17716.457,E2 -17716.457} C_VEL
LIN {X 0,Y 269.354,Z 362.239,A -85,B 0,C 180,E1 -17718.717,E2 -17718.717} C_VEL
LIN {X 0,Y 268.971,Z 369.988,A -85,B 0,C 180,E1 -17720.982,E2 -17720.982} C_VEL
LIN {X 0,Y 268.817,Z 376.654,A -85,B 0,C 180,E1 -17723.454,E2 -17723.454} C_VEL
LIN {X 0,Y 268.737,Z 380.996,A -85,B 0,C 180,E1 -17725.502,E2 -17725.502} C_VEL
LIN {X 0,Y 268.839,Z 384.644,A -85,B 0,C 180,E1 -17727.755,E2 -17727.755} C_VEL
LIN {X 0,Y 268.868,Z 387.202,A -85,B 0,C 180,E1 -17730.002,E2 -17730.002} C_VEL
LIN {X 0,Y 268.769,Z 388.321,A -85,B 0,C 180,E1 -17731.5,E2 -17731.5} C_VEL
LIN {X 0,Y 268.404,Z 389.327,A -85,B 0,C 180,E1 -17734.507,E2 -17734.507} C_VEL
LIN {X 0,Y 268.477,Z 388.706,A -85,B 0,C 180,E1 -17737.523,E2 -17737.523} C_VEL
LIN {X 0,Y 269.208,Z 386.582,A -85,B 0,C 180,E1 -17740.531,E2 -17740.531} C_VEL
LIN {X 0,Y 270.575,Z 382.92,A -85,B 0,C 180,E1 -17743.521,E2 -17743.521} C_VEL
LIN {X 0,Y 273.063,Z 377.66,A -85,B 0,C 180,E1 -17746.448,E2 -17746.448} C_VEL
LIN {X 0,Y 275.163,Z 372.611,A -85,B 0,C 180,E1 -17748.62,E2 -17748.62} C_VEL
LIN {X 0,Y 278.375,Z 365.396,A -85,B 0,C 180,E1 -17751.087,E2 -17751.087} C_VEL
LIN {X 0,Y 282.491,Z 356.475,A -85,B 0,C 180,E1 -17753.459,E2 -17753.459} C_VEL
LIN {X 0,Y 286.51,Z 347.318,A -85,B 0,C 180,E1 -17755.423,E2 -17755.423} C_VEL
LIN {X 0,Y 291.646,Z 334.401,A -85,B 0,C 180,E1 -17757.64,E2 -17757.64} C_VEL
LIN {X 0,Y 295.129,Z 322.634,A -85,B 0,C 180,E1 -17759.418,E2 -17759.418} C_VEL
LIN {X 0,Y 297.229,Z 311.633,A -85,B 0,C 180,E1 -17761.058,E2 -17761.058} C_VEL
LIN {X 0,Y 298.228,Z 300.532,A -85,B 0,C 180,E1 -17762.823,E2 -17762.823} C_VEL
LIN {X 0,Y 298.456,Z 288.877,A -85,B 0,C 180,E1 -17764.825,E2 -17764.825} C_VEL
LIN {X 0,Y 298.02,Z 279.464,A -85,B 0,C 180,E1 -17766.698,E2 -17766.698} C_VEL
LIN {X 0,Y 297.61,Z 277.477,A -85,B 0,C 180,E1 -17767.293,E2 -17767.293} C_VEL
LIN {X 0,Y 296.589,Z 274.221,A -85,B 0,C 180,E1 -17768.558,E2 -17768.558} C_VEL
LIN {X 0,Y 295.168,Z 271.271,A -85,B 0,C 180,E1 -17770.366,E2 -17770.366} C_VEL
LIN {X 0,Y 294.057,Z 269.506,A -85,B 0,C 180,E1 -17772.191,E2 -17772.191} C_VEL
LIN {X 0,Y 293.257,Z 268.899,A -85,B 0,C 180,E1 -17774.031,E2 -17774.031} C_VEL
LIN {X 0,Y 292.859,Z 269.222,A -85,B 0,C 180,E1 -17776.051,E2 -17776.051} C_VEL
LIN {X 0,Y 293.064,Z 270.188,A -85,B 0,C 180,E1 -17778.025,E2 -17778.025} C_VEL
LIN {X 0,Y 293.634,Z 272.327,A -85,B 0,C 180,E1 -17779.99,E2 -17779.99} C_VEL
LIN {X 0,Y 294.386,Z 274.958,A -85,B 0,C 180,E1 -17781.632,E2 -17781.632} C_VEL
LIN {X 0,Y 295.329,Z 281.027,A -85,B 0,C 180,E1 -17784.011,E2 -17784.011} C_VEL
LIN {X 0,Y 296.551,Z 288.147,A -85,B 0,C 180,E1 -17786.386,E2 -17786.386} C_VEL
LIN {X 0,Y 297.796,Z 297.736,A -85,B 0,C 180,E1 -17789.116,E2 -17789.116} C_VEL
LIN {X 0,Y 298.05,Z 306.381,A -85,B 0,C 180,E1 -17791.239,E2 -17791.239} C_VEL
LIN {X 0,Y 297.921,Z 309.089,A -85,B 0,C 180,E1 -17791.849,E2 -17791.849} C_VEL
LIN {X 0,Y 293.46,Z 320.669,A -85,B 0,C 180,E1 -17793.701,E2 -17793.701} C_VEL
LIN {X 0,Y 289.274,Z 330.253,A -85,B 0,C 180,E1 -17795.605,E2 -17795.605} C_VEL
LIN {X 0,Y 284.828,Z 339.454,A -85,B 0,C 180,E1 -17797.896,E2 -17797.896} C_VEL
LIN {X 0,Y 280.953,Z 346.798,A -85,B 0,C 180,E1 -17800.263,E2 -17800.263} C_VEL
LIN {X 0,Y 278.12,Z 351.876,A -85,B 0,C 180,E1 -17802.348,E2 -17802.348} C_VEL
LIN {X 0,Y 275.746,Z 355.921,A -85,B 0,C 180,E1 -17804.478,E2 -17804.478} C_VEL
LIN {X 0,Y 273.691,Z 359.047,A -85,B 0,C 180,E1 -17806.638,E2 -17806.638} C_VEL
LIN {X 0,Y 271.603,Z 361.845,A -85,B 0,C 180,E1 -17809.564,E2 -17809.564} C_VEL
LIN {X 0,Y 270.554,Z 362.668,A -85,B 0,C 180,E1 -17811.033,E2 -17811.033} C_VEL
LIN {X 0,Y 269.504,Z 363.15,A -85,B 0,C 180,E1 -17814.013,E2 -17814.013} C_VEL
LIN {X 0,Y 269.127,Z 362.84,A -85,B 0,C 180,E1 -17815.507,E2 -17815.507} C_VEL
LIN {X 0,Y 268.533,Z 360.998,A -85,B 0,C 180,E1 -17818.5,E2 -17818.5} C_VEL
LIN {X 0,Y 268.387,Z 357.582,A -85,B 0,C 180,E1 -17821.501,E2 -17821.501} C_VEL
LIN {X 0,Y 268.516,Z 353.872,A -85,B 0,C 180,E1 -17823.752,E2 -17823.752} C_VEL
LIN {X 0,Y 268.623,Z 348.659,A -85,B 0,C 180,E1 -17826.164,E2 -17826.164} C_VEL
LIN {X 0,Y 269.092,Z 341.887,A -85,B 0,C 180,E1 -17828.637,E2 -17828.637} C_VEL
LIN {X 0,Y 269.719,Z 334.232,A -85,B 0,C 180,E1 -17830.889,E2 -17830.889} C_VEL
LIN {X 0,Y 270.549,Z 324.753,A -85,B 0,C 180,E1 -17833.138,E2 -17833.138} C_VEL
LIN {X 0,Y 271.694,Z 314.187,A -85,B 0,C 180,E1 -17835.183,E2 -17835.183} C_VEL
LIN {X 0,Y 272.716,Z 302.749,A -85,B 0,C 180,E1 -17836.98,E2 -17836.98} C_VEL
LIN {X 0,Y 273.809,Z 290.519,A -85,B 0,C 180,E1 -17838.52,E2 -17838.52} C_VEL
LIN {X 0,Y 274.339,Z 280.595,A -85,B 0,C 180,E1 -17839.541,E2 -17839.541} C_VEL
LIN {X 0,Y 272.126,Z 266.222,A -85,B 0,C 180,E1 -17840.793,E2 -17840.793} C_VEL
LIN {X 0,Y 270.425,Z 252.968,A -85,B 0,C 180,E1 -17841.687,E2 -17841.687} C_VEL
LIN {X 0,Y 270.923,Z 245.232,A -85,B 0,C 180,E1 -17845.362,E2 -17845.362} C_VEL
LIN {X 0,Y 271.38,Z 236.675,A -85,B 0,C 180,E1 -17849.476,E2 -17849.476} C_VEL
LIN {X 0,Y 271.909,Z 229.614,A -85,B 0,C 180,E1 -17852.874,E2 -17852.874} C_VEL
LIN {X 0,Y 272.223,Z 224.194,A -85,B 0,C 180,E1 -17855.513,E2 -17855.513} C_VEL
LIN {X 0,Y 272.079,Z 220.193,A -85,B 0,C 180,E1 -17857.505,E2 -17857.505} C_VEL
LIN {X 0,Y 271.133,Z 214.56,A -85,B 0,C 180,E1 -17860.393,E2 -17860.393} C_VEL
LIN {X 0,Y 270.252,Z 209.823,A -85,B 0,C 180,E1 -17862.877,E2 -17862.877} C_VEL
LIN {X 0,Y 270.178,Z 209.829,A -85,B 0,C 180,E1 -17867.441,E2 -17867.441} C_VEL
LIN {X 0,Y 270.213,Z 209.829,A -85,B 0,C 180,E1 -17871.373,E2 -17871.373} C_VEL
LIN {X 0,Y 270.26,Z 209.901,A -85,B 0,C 180,E1 -17873.413,E2 -17873.413} C_VEL
LIN {X 0,Y 270.741,Z 213.038,A -85,B 0,C 180,E1 -17876.965,E2 -17876.965} C_VEL
LIN {X 0,Y 270.973,Z 216.39,A -85,B 0,C 180,E1 -17880.474,E2 -17880.474} C_VEL
LIN {X 0,Y 270.87,Z 219.785,A -85,B 0,C 180,E1 -17883.825,E2 -17883.825} C_VEL
LIN {X 0,Y 270.729,Z 223.279,A -85,B 0,C 180,E1 -17887.081,E2 -17887.081} C_VEL
LIN {X 0,Y 270.638,Z 226.894,A -85,B 0,C 180,E1 -17890.268,E2 -17890.268} C_VEL
LIN {X 0,Y 270.637,Z 227.989,A -85,B 0,C 180,E1 -17891.204,E2 -17891.204} C_VEL
LIN {X 0,Y 273.981,Z 239.151,A -85,B 0,C 180,E1 -17892.174,E2 -17892.174} C_VEL
LIN {X 0,Y 276.371,Z 248.864,A -85,B 0,C 180,E1 -17893.264,E2 -17893.264} C_VEL
LIN {X 0,Y 277.459,Z 256.369,A -85,B 0,C 180,E1 -17894.268,E2 -17894.268} C_VEL
LIN {X 0,Y 276.627,Z 264.431,A -85,B 0,C 180,E1 -17895.468,E2 -17895.468} C_VEL
LIN {X 0,Y 275.693,Z 271.154,A -85,B 0,C 180,E1 -17896.735,E2 -17896.735} C_VEL
LIN {X 0,Y 274.55,Z 277.412,A -85,B 0,C 180,E1 -17898.181,E2 -17898.181} C_VEL
LIN {X 0,Y 273.557,Z 282.347,A -85,B 0,C 180,E1 -17899.638,E2 -17899.638} C_VEL
LIN {X 0,Y 272.694,Z 286.31,A -85,B 0,C 180,E1 -17901.103,E2 -17901.103} C_VEL
LIN {X 0,Y 272.127,Z 290.711,A -85,B 0,C 180,E1 -17903.324,E2 -17903.324} C_VEL
LIN {X 0,Y 271.228,Z 293.703,A -85,B 0,C 180,E1 -17905.54,E2 -17905.54} C_VEL
LIN {X 0,Y 271.028,Z 294.958,A -85,B 0,C 180,E1 -17907.025,E2 -17907.025} C_VEL
LIN {X 0,Y 270.81,Z 295.722,A -85,B 0,C 180,E1 -17908.511,E2 -17908.511} C_VEL
LIN {X 0,Y 270.722,Z 295.991,A -85,B 0,C 180,E1 -17909.998,E2 -17909.998} C_VEL
LIN {X 0,Y 270.808,Z 295.758,A -85,B 0,C 180,E1 -17911.485,E2 -17911.485} C_VEL
LIN {X 0,Y 271.025,Z 295.042,A -85,B 0,C 180,E1 -17912.971,E2 -17912.971} C_VEL
LIN {X 0,Y 271.225,Z 293.838,A -85,B 0,C 180,E1 -17914.456,E2 -17914.456} C_VEL
LIN {X 0,Y 272.117,Z 290.913,A -85,B 0,C 180,E1 -17916.672,E2 -17916.672} C_VEL
LIN {X 0,Y 272.655,Z 286.597,A -85,B 0,C 180,E1 -17918.895,E2 -17918.895} C_VEL
LIN {X 0,Y 273.398,Z 283.746,A -85,B 0,C 180,E1 -17919.99,E2 -17919.99} C_VEL
LIN {X 0,Y 274.258,Z 279.155,A -85,B 0,C 180,E1 -17921.453,E2 -17921.453} C_VEL
LIN {X 0,Y 275.386,Z 273.383,A -85,B 0,C 180,E1 -17922.901,E2 -17922.901} C_VEL
LIN {X 0,Y 276.307,Z 267.146,A -85,B 0,C 180,E1 -17924.169,E2 -17924.169} C_VEL
LIN {X 0,Y 277.084,Z 259.874,A -85,B 0,C 180,E1 -17925.36,E2 -17925.36} C_VEL
LIN {X 0,Y 277.464,Z 255.197,A -85,B 0,C 180,E1 -17926.01,E2 -17926.01} C_VEL
LIN {X 0,Y 275.837,Z 246.354,A -85,B 0,C 180,E1 -17927.167,E2 -17927.167} C_VEL
LIN {X 0,Y 273.19,Z 236.21,A -85,B 0,C 180,E1 -17928.226,E2 -17928.226} C_VEL
LIN {X 0,Y 270.629,Z 227.988,A -85,B 0,C 180,E1 -17928.939,E2 -17928.939} C_VEL
LIN {X 0,Y 270.737,Z 223.44,A -85,B 0,C 180,E1 -17932.914,E2 -17932.914} C_VEL
LIN {X 0,Y 270.878,Z 219.966,A -85,B 0,C 180,E1 -17936.17,E2 -17936.17} C_VEL
LIN {X 0,Y 270.974,Z 216.55,A -85,B 0,C 180,E1 -17939.521,E2 -17939.521} C_VEL
LIN {X 0,Y 270.723,Z 213.174,A -85,B 0,C 180,E1 -17943.033,E2 -17943.033} C_VEL
LIN {X 0,Y 270.232,Z 209.825,A -85,B 0,C 180,E1 -17946.969,E2 -17946.969} C_VEL
LIN {X 0,Y 270.164,Z 209.832,A -85,B 0,C 180,E1 -17951.027,E2 -17951.027} C_VEL
LIN {X 0,Y 270.165,Z 209.833,A -85,B 0,C 180,E1 -17955.382,E2 -17955.382} C_VEL
LIN {X 0,Y 270.179,Z 209.825,A -85,B 0,C 180,E1 -17959.435,E2 -17959.435} C_VEL
LIN {X 0,Y 270.212,Z 209.821,A -85,B 0,C 180,E1 -17963.258,E2 -17963.258} C_VEL
LIN {X 0,Y 270.195,Z 209.822,A -85,B 0,C 180,E1 -17966.891,E2 -17966.891} C_VEL
LIN {X 0,Y 270.22,Z 209.816,A -85,B 0,C 180,E1 -17970.385,E2 -17970.385} C_VEL
LIN {X 0,Y 270.255,Z 209.816,A -85,B 0,C 180,E1 -17973.763,E2 -17973.763} C_VEL
LIN {X 0,Y 270.224,Z 209.824,A -85,B 0,C 180,E1 -17977.038,E2 -17977.038} C_VEL
LIN {X 0,Y 270.292,Z 209.805,A -85,B 0,C 180,E1 -17980.244,E2 -17980.244} C_VEL
LIN {X 0,Y 270.393,Z 209.789,A -85,B 0,C 180,E1 -17984.935,E2 -17984.935} C_VEL
LIN {X 0,Y 270.402,Z 209.789,A -85,B 0,C 180,E1 -17989.517,E2 -17989.517} C_VEL
LIN {X 0,Y 270.588,Z 209.778,A -85,B 0,C 180,E1 -17992.538,E2 -17992.538} C_VEL
LIN {X 0,Y 270.776,Z 209.752,A -85,B 0,C 180,E1 -17998.513,E2 -17998.513} C_VEL
LIN {X 0,Y 270.775,Z 209.752,A -85,B 0,C 180,E1 -18001.487,E2 -18001.487} C_VEL
LIN {X 0,Y 270.6,Z 209.777,A -85,B 0,C 180,E1 -18007.461,E2 -18007.461} C_VEL
LIN {X 0,Y 270.431,Z 209.794,A -85,B 0,C 180,E1 -18010.481,E2 -18010.481} C_VEL
LIN {X 0,Y 270.379,Z 209.801,A -85,B 0,C 180,E1 -18011.507,E2 -18011.507} C_VEL
LIN {X 0,Y 269.694,Z 209.891,A -85,B 0,C 180,E1 -18012.751,E2 -18012.751} C_VEL
LIN {X 0,Y 266.774,Z 210.252,A -85,B 0,C 180,E1 -18014.776,E2 -18014.776} C_VEL
LIN {X 0,Y 264.3,Z 210.559,A -85,B 0,C 180,E1 -18016.422,E2 -18016.422} C_VEL
LIN {X 0,Y 263.247,Z 210.686,A -85,B 0,C 180,E1 -18017.7,E2 -18017.7} C_VEL
LIN {X 0,Y 263.165,Z 210.697,A -85,B 0,C 180,E1 -18018.134,E2 -18018.134} C_VEL
LIN {X 0,Y 263.163,Z 210.706,A -85,B 0,C 180,E1 -18020.826,E2 -18020.826} C_VEL
LIN {X 0,Y 263.117,Z 210.714,A -85,B 0,C 180,E1 -18025.301,E2 -18025.301} C_VEL
LIN {X 0,Y 263.122,Z 210.712,A -85,B 0,C 180,E1 -18028.736,E2 -18028.736} C_VEL
LIN {X 0,Y 263.119,Z 210.709,A -85,B 0,C 180,E1 -18032.29,E2 -18032.29} C_VEL
LIN {X 0,Y 263.171,Z 210.756,A -85,B 0,C 180,E1 -18035.863,E2 -18035.863} C_VEL
LIN {X 0,Y 264.547,Z 216.379,A -85,B 0,C 180,E1 -18039.612,E2 -18039.612} C_VEL
LIN {X 0,Y 265.954,Z 222.56,A -85,B 0,C 180,E1 -18043.398,E2 -18043.398} C_VEL
LIN {X 0,Y 267.605,Z 229.718,A -85,B 0,C 180,E1 -18047.337,E2 -18047.337} C_VEL
LIN {X 0,Y 269.334,Z 237.414,A -85,B 0,C 180,E1 -18051.228,E2 -18051.228} C_VEL
LIN {X 0,Y 271.095,Z 246.037,A -85,B 0,C 180,E1 -18055.229,E2 -18055.229} C_VEL
LIN {X 0,Y 271.323,Z 247.752,A -85,B 0,C 180,E1 -18055.985,E2 -18055.985} C_VEL
LIN {X 0,Y 268.595,Z 257.17,A -85,B 0,C 180,E1 -18059.709,E2 -18059.709} C_VEL
LIN {X 0,Y 265.704,Z 268.953,A -85,B 0,C 180,E1 -18064.439,E2 -18064.439} C_VEL
LIN {X 0,Y 265.227,Z 271.295,A -85,B 0,C 180,E1 -18065.335,E2 -18065.335} C_VEL
LIN {X 0,Y 266.436,Z 283.999,A -85,B 0,C 180,E1 -18066.102,E2 -18066.102} C_VEL
LIN {X 0,Y 266.867,Z 296.21,A -85,B 0,C 180,E1 -18067.119,E2 -18067.119} C_VEL
LIN {X 0,Y 266.84,Z 307.758,A -85,B 0,C 180,E1 -18068.365,E2 -18068.365} C_VEL
LIN {X 0,Y 266.83,Z 317.984,A -85,B 0,C 180,E1 -18069.778,E2 -18069.778} C_VEL
LIN {X 0,Y 266.243,Z 325.293,A -85,B 0,C 180,E1 -18070.936,E2 -18070.936} C_VEL
LIN {X 0,Y 264.98,Z 333.78,A -85,B 0,C 180,E1 -18072.533,E2 -18072.533} C_VEL
LIN {X 0,Y 263.841,Z 342.574,A -85,B 0,C 180,E1 -18074.554,E2 -18074.554} C_VEL
LIN {X 0,Y 262.853,Z 353.925,A -85,B 0,C 180,E1 -18076.866,E2 -18076.866} C_VEL
LIN {X 0,Y 262.174,Z 363.196,A -85,B 0,C 180,E1 -18079.187,E2 -18079.187} C_VEL
LIN {X 0,Y 261.884,Z 370.623,A -85,B 0,C 180,E1 -18081.514,E2 -18081.514} C_VEL
LIN {X 0,Y 261.762,Z 376.544,A -85,B 0,C 180,E1 -18083.837,E2 -18083.837} C_VEL
LIN {X 0,Y 261.752,Z 381.172,A -85,B 0,C 180,E1 -18086.153,E2 -18086.153} C_VEL
LIN {X 0,Y 261.844,Z 384.626,A -85,B 0,C 180,E1 -18088.464,E2 -18088.464} C_VEL
LIN {X 0,Y 261.831,Z 386.334,A -85,B 0,C 180,E1 -18090.002,E2 -18090.002} C_VEL
LIN {X 0,Y 261.705,Z 387.569,A -85,B 0,C 180,E1 -18091.541,E2 -18091.541} C_VEL
LIN {X 0,Y 261.325,Z 388.748,A -85,B 0,C 180,E1 -18094.63,E2 -18094.63} C_VEL
LIN {X 0,Y 261.404,Z 388.404,A -85,B 0,C 180,E1 -18097.727,E2 -18097.727} C_VEL
LIN {X 0,Y 262.189,Z 386.498,A -85,B 0,C 180,E1 -18100.817,E2 -18100.817} C_VEL
LIN {X 0,Y 263.662,Z 383.128,A -85,B 0,C 180,E1 -18103.882,E2 -18103.882} C_VEL
LIN {X 0,Y 265.565,Z 379.565,A -85,B 0,C 180,E1 -18106.135,E2 -18106.135} C_VEL
LIN {X 0,Y 267.736,Z 375.096,A -85,B 0,C 180,E1 -18108.362,E2 -18108.362} C_VEL
LIN {X 0,Y 270.599,Z 369.061,A -85,B 0,C 180,E1 -18110.772,E2 -18110.772} C_VEL
LIN {X 0,Y 274.213,Z 361.967,A -85,B 0,C 180,E1 -18113.009,E2 -18113.009} C_VEL
LIN {X 0,Y 278.852,Z 352.501,A -85,B 0,C 180,E1 -18115.371,E2 -18115.371} C_VEL
LIN {X 0,Y 283.352,Z 342.803,A -85,B 0,C 180,E1 -18117.315,E2 -18117.315} C_VEL
LIN {X 0,Y 287.545,Z 332.404,A -85,B 0,C 180,E1 -18119.065,E2 -18119.065} C_VEL
LIN {X 0,Y 290.82,Z 321.674,A -85,B 0,C 180,E1 -18120.754,E2 -18120.754} C_VEL
LIN {X 0,Y 292.93,Z 311.219,A -85,B 0,C 180,E1 -18122.429,E2 -18122.429} C_VEL
LIN {X 0,Y 294.129,Z 300.548,A -85,B 0,C 180,E1 -18124.254,E2 -18124.254} C_VEL
LIN {X 0,Y 294.602,Z 290.801,A -85,B 0,C 180,E1 -18126.103,E2 -18126.103} C_VEL
LIN {X 0,Y 294.654,Z 284.325,A -85,B 0,C 180,E1 -18127.481,E2 -18127.481} C_VEL
LIN {X 0,Y 294.123,Z 281.729,A -85,B 0,C 180,E1 -18128.41,E2 -18128.41} C_VEL
LIN {X 0,Y 293.128,Z 278.777,A -85,B 0,C 180,E1 -18129.894,E2 -18129.894} C_VEL
LIN {X 0,Y 291.976,Z 276.653,A -85,B 0,C 180,E1 -18131.739,E2 -18131.739} C_VEL
LIN {X 0,Y 291.093,Z 275.755,A -85,B 0,C 180,E1 -18133.589,E2 -18133.589} C_VEL
LIN {X 0,Y 290.577,Z 275.79,A -85,B 0,C 180,E1 -18135.46,E2 -18135.46} C_VEL
LIN {X 0,Y 290.542,Z 276.533,A -85,B 0,C 180,E1 -18137.367,E2 -18137.367} C_VEL
LIN {X 0,Y 290.85,Z 278.197,A -85,B 0,C 180,E1 -18139.276,E2 -18139.276} C_VEL
LIN {X 0,Y 291.392,Z 280.971,A -85,B 0,C 180,E1 -18141.164,E2 -18141.164} C_VEL
LIN {X 0,Y 291.933,Z 287.278,A -85,B 0,C 180,E1 -18143.762,E2 -18143.762} C_VEL
LIN {X 0,Y 292.693,Z 295.281,A -85,B 0,C 180,E1 -18146.477,E2 -18146.477} C_VEL
LIN {X 0,Y 293.172,Z 302.319,A -85,B 0,C 180,E1 -18148.574,E2 -18148.574} C_VEL
LIN {X 0,Y 292.94,Z 310.452,A -85,B 0,C 180,E1 -18150.689,E2 -18150.689} C_VEL
LIN {X 0,Y 292.817,Z 311.7,A -85,B 0,C 180,E1 -18150.995,E2 -18150.995} C_VEL
LIN {X 0,Y 288.344,Z 322.462,A -85,B 0,C 180,E1 -18152.806,E2 -18152.806} C_VEL
LIN {X 0,Y 283.906,Z 331.755,A -85,B 0,C 180,E1 -18154.722,E2 -18154.722} C_VEL
LIN {X 0,Y 279.193,Z 340.686,A -85,B 0,C 180,E1 -18157.035,E2 -18157.035} C_VEL
LIN {X 0,Y 275.616,Z 346.926,A -85,B 0,C 180,E1 -18159.085,E2 -18159.085} C_VEL
LIN {X 0,Y 272.506,Z 352.042,A -85,B 0,C 180,E1 -18161.193,E2 -18161.193} C_VEL
LIN {X 0,Y 269.792,Z 356.161,A -85,B 0,C 180,E1 -18163.349,E2 -18163.349} C_VEL
LIN {X 0,Y 266.885,Z 360.208,A -85,B 0,C 180,E1 -18166.29,E2 -18166.29} C_VEL
LIN {X 0,Y 264.803,Z 362.574,A -85,B 0,C 180,E1 -18169.119,E2 -18169.119} C_VEL
LIN {X 0,Y 263.595,Z 363.375,A -85,B 0,C 180,E1 -18170.795,E2 -18170.795} C_VEL
LIN {X 0,Y 262.465,Z 363.613,A -85,B 0,C 180,E1 -18173.851,E2 -18173.851} C_VEL
LIN {X 0,Y 262.068,Z 363.141,A -85,B 0,C 180,E1 -18175.385,E2 -18175.385} C_VEL
LIN {X 0,Y 261.453,Z 361.086,A -85,B 0,C 180,E1 -18178.46,E2 -18178.46} C_VEL
LIN {X 0,Y 261.288,Z 358.476,A -85,B 0,C 180,E1 -18180.771,E2 -18180.771} C_VEL
LIN {X 0,Y 261.415,Z 354.909,A -85,B 0,C 180,E1 -18183.082,E2 -18183.082} C_VEL
LIN {X 0,Y 261.473,Z 350.068,A -85,B 0,C 180,E1 -18185.492,E2 -18185.492} C_VEL
LIN {X 0,Y 261.911,Z 343.36,A -85,B 0,C 180,E1 -18188.099,E2 -18188.099} C_VEL
LIN {X 0,Y 262.485,Z 335.925,A -85,B 0,C 180,E1 -18190.412,E2 -18190.412} C_VEL
LIN {X 0,Y 263.281,Z 326.816,A -85,B 0,C 180,E1 -18192.722,E2 -18192.722} C_VEL
LIN {X 0,Y 264.463,Z 315.61,A -85,B 0,C 180,E1 -18195.017,E2 -18195.017} C_VEL
LIN {X 0,Y 265.468,Z 305.252,A -85,B 0,C 180,E1 -18196.733,E2 -18196.733} C_VEL
LIN {X 0,Y 266.408,Z 294.165,A -85,B 0,C 180,E1 -18198.245,E2 -18198.245} C_VEL
LIN {X 0,Y 267.402,Z 282.088,A -85,B 0,C 180,E1 -18199.579,E2 -18199.579} C_VEL
LIN {X 0,Y 265.123,Z 267.051,A -85,B 0,C 180,E1 -18200.941,E2 -18200.941} C_VEL
LIN {X 0,Y 263.398,Z 253.35,A -85,B 0,C 180,E1 -18201.882,E2 -18201.882} C_VEL
LIN {X 0,Y 263.919,Z 244.684,A -85,B 0,C 180,E1 -18206.065,E2 -18206.065} C_VEL
LIN {X 0,Y 264.457,Z 235.945,A -85,B 0,C 180,E1 -18210.327,E2 -18210.327} C_VEL
LIN {X 0,Y 264.964,Z 228.76,A -85,B 0,C 180,E1 -18213.85,E2 -18213.85} C_VEL
LIN {X 0,Y 265.244,Z 223.462,A -85,B 0,C 180,E1 -18216.472,E2 -18216.472} C_VEL
LIN {X 0,Y 264.46,Z 217.358,A -85,B 0,C 180,E1 -18219.628,E2 -18219.628} C_VEL
LIN {X 0,Y 263.191,Z 210.702,A -85,B 0,C 180,E1 -18223.168,E2 -18223.168} C_VEL
LIN {X 0,Y 263.13,Z 210.71,A -85,B 0,C 180,E1 -18226.15,E2 -18226.15} C_VEL
LIN {X 0,Y 263.111,Z 210.714,A -85,B 0,C 180,E1 -18230.126,E2 -18230.126} C_VEL
LIN {X 0,Y 263.207,Z 210.923,A -85,B 0,C 180,E1 -18232.743,E2 -18232.743} C_VEL
LIN {X 0,Y 263.702,Z 213.686,A -85,B 0,C 180,E1 -18235.965,E2 -18235.965} C_VEL
LIN {X 0,Y 263.983,Z 217.028,A -85,B 0,C 180,E1 -18239.611,E2 -18239.611} C_VEL
LIN {X 0,Y 263.933,Z 220.468,A -85,B 0,C 180,E1 -18243.083,E2 -18243.083} C_VEL
LIN {X 0,Y 263.806,Z 223.984,A -85,B 0,C 180,E1 -18246.444,E2 -18246.444} C_VEL
LIN {X 0,Y 263.673,Z 228.638,A -85,B 0,C 180,E1 -18250.612,E2 -18250.612} C_VEL
LIN {X 0,Y 267.025,Z 239.472,A -85,B 0,C 180,E1 -18251.587,E2 -18251.587} C_VEL
LIN {X 0,Y 269.591,Z 250.103,A -85,B 0,C 180,E1 -18252.816,E2 -18252.816} C_VEL
LIN {X 0,Y 270.728,Z 257.43,A -85,B 0,C 180,E1 -18253.844,E2 -18253.844} C_VEL
LIN {X 0,Y 269.842,Z 265.535,A -85,B 0,C 180,E1 -18255.095,E2 -18255.095} C_VEL
LIN {X 0,Y 268.872,Z 272.212,A -85,B 0,C 180,E1 -18256.392,E2 -18256.392} C_VEL
LIN {X 0,Y 267.683,Z 278.44,A -85,B 0,C 180,E1 -18257.873,E2 -18257.873} C_VEL
LIN {X 0,Y 266.647,Z 283.35,A -85,B 0,C 180,E1 -18259.366,E2 -18259.366} C_VEL
LIN {X 0,Y 265.751,Z 287.3,A -85,B 0,C 180,E1 -18260.868,E2 -18260.868} C_VEL
LIN {X 0,Y 265.148,Z 291.692,A -85,B 0,C 180,E1 -18263.148,E2 -18263.148} C_VEL
LIN {X 0,Y 264.223,Z 294.679,A -85,B 0,C 180,E1 -18265.421,E2 -18265.421} C_VEL
LIN {X 0,Y 264.011,Z 295.932,A -85,B 0,C 180,E1 -18266.946,E2 -18266.946} C_VEL
LIN {X 0,Y 263.785,Z 296.696,A -85,B 0,C 180,E1 -18268.471,E2 -18268.471} C_VEL
LIN {X 0,Y 263.695,Z 296.965,A -85,B 0,C 180,E1 -18269.998,E2 -18269.998} C_VEL
LIN {X 0,Y 263.783,Z 296.731,A -85,B 0,C 180,E1 -18271.525,E2 -18271.525} C_VEL
LIN {X 0,Y 264.008,Z 296.016,A -85,B 0,C 180,E1 -18273.05,E2 -18273.05} C_VEL
LIN {X 0,Y 264.22,Z 294.813,A -85,B 0,C 180,E1 -18274.575,E2 -18274.575} C_VEL
LIN {X 0,Y 265.137,Z 291.89,A -85,B 0,C 180,E1 -18276.849,E2 -18276.849} C_VEL
LIN {X 0,Y 265.711,Z 287.583,A -85,B 0,C 180,E1 -18279.129,E2 -18279.129} C_VEL
LIN {X 0,Y 266.479,Z 284.746,A -85,B 0,C 180,E1 -18280.252,E2 -18280.252} C_VEL
LIN {X 0,Y 267.376,Z 280.179,A -85,B 0,C 180,E1 -18281.752,E2 -18281.752} C_VEL
LIN {X 0,Y 268.551,Z 274.436,A -85,B 0,C 180,E1 -18283.235,E2 -18283.235} C_VEL
LIN {X 0,Y 269.641,Z 267.228,A -85,B 0,C 180,E1 -18284.72,E2 -18284.72} C_VEL
LIN {X 0,Y 270.358,Z 260.906,A -85,B 0,C 180,E1 -18285.771,E2 -18285.771} C_VEL
LIN {X 0,Y 270.694,Z 256.347,A -85,B 0,C 180,E1 -18286.433,E2 -18286.433} C_VEL
LIN {X 0,Y 269.109,Z 247.724,A -85,B 0,C 180,E1 -18287.61,E2 -18287.61} C_VEL
LIN {X 0,Y 266.708,Z 238.41,A -85,B 0,C 180,E1 -18288.645,E2 -18288.645} C_VEL
LIN {X 0,Y 263.663,Z 228.608,A -85,B 0,C 180,E1 -18289.561,E2 -18289.561} C_VEL
LIN {X 0,Y 263.816,Z 224.147,A -85,B 0,C 180,E1 -18293.551,E2 -18293.551} C_VEL
LIN {X 0,Y 263.939,Z 220.627,A -85,B 0,C 180,E1 -18296.912,E2 -18296.912} C_VEL
LIN {X 0,Y 263.978,Z 217.218,A -85,B 0,C 180,E1 -18300.385,E2 -18300.385} C_VEL
LIN {X 0,Y 263.663,Z 213.587,A -85,B 0,C 180,E1 -18304.278,E2 -18304.278} C_VEL
LIN {X 0,Y 263.183,Z 210.702,A -85,B 0,C 180,E1 -18307.89,E2 -18307.89} C_VEL
LIN {X 0,Y 263.119,Z 210.708,A -85,B 0,C 180,E1 -18311.891,E2 -18311.891} C_VEL
LIN {X 0,Y 263.128,Z 210.705,A -85,B 0,C 180,E1 -18316.147,E2 -18316.147} C_VEL
LIN {X 0,Y 263.115,Z 210.707,A -85,B 0,C 180,E1 -18320.129,E2 -18320.129} C_VEL
LIN {X 0,Y 263.156,Z 210.704,A -85,B 0,C 180,E1 -18324.017,E2 -18324.017} C_VEL
LIN {X 0,Y 263.125,Z 210.707,A -85,B 0,C 180,E1 -18327.71,E2 -18327.71} C_VEL
LIN {X 0,Y 263.192,Z 210.697,A -85,B 0,C 180,E1 -18331.782,E2 -18331.782} C_VEL
LIN {X 0,Y 263.217,Z 210.685,A -85,B 0,C 180,E1 -18335.199,E2 -18335.199} C_VEL
LIN {X 0,Y 263.254,Z 210.681,A -85,B 0,C 180,E1 -18339.692,E2 -18339.692} C_VEL
LIN {X 0,Y 263.341,Z 210.668,A -85,B 0,C 180,E1 -18344.521,E2 -18344.521} C_VEL
LIN {X 0,Y 263.345,Z 210.67,A -85,B 0,C 180,E1 -18349.233,E2 -18349.233} C_VEL
LIN {X 0,Y 263.547,Z 210.654,A -85,B 0,C 180,E1 -18352.338,E2 -18352.338} C_VEL
LIN {X 0,Y 263.741,Z 210.629,A -85,B 0,C 180,E1 -18358.473,E2 -18358.473} C_VEL
LIN {X 0,Y 263.74,Z 210.628,A -85,B 0,C 180,E1 -18361.527,E2 -18361.527} C_VEL
LIN {X 0,Y 263.562,Z 210.654,A -85,B 0,C 180,E1 -18367.662,E2 -18367.662} C_VEL
LIN {X 0,Y 263.363,Z 210.678,A -85,B 0,C 180,E1 -18370.766,E2 -18370.766} C_VEL
LIN {X 0,Y 263.3,Z 210.688,A -85,B 0,C 180,E1 -18375.481,E2 -18375.481} C_VEL
LIN {X 0,Y 263.165,Z 210.697,A -85,B 0,C 180,E1 -18378.134,E2 -18378.134} C_VEL
LIN {X 0,Y 262.5,Z 210.789,A -85,B 0,C 180,E1 -18379.411,E2 -18379.411} C_VEL
LIN {X 0,Y 259.619,Z 211.149,A -85,B 0,C 180,E1 -18381.492,E2 -18381.492} C_VEL
LIN {X 0,Y 257.179,Z 211.453,A -85,B 0,C 180,E1 -18383.185,E2 -18383.185} C_VEL
LIN {X 0,Y 256.148,Z 211.58,A -85,B 0,C 180,E1 -18384.499,E2 -18384.499} C_VEL
LIN {X 0,Y 256.072,Z 211.59,A -85,B 0,C 180,E1 -18384.944,E2 -18384.944} C_VEL
LIN {X 0,Y 256.079,Z 211.589,A -85,B 0,C 180,E1 -18388.576,E2 -18388.576} C_VEL
LIN {X 0,Y 256.065,Z 211.59,A -85,B 0,C 180,E1 -18391.703,E2 -18391.703} C_VEL
LIN {X 0,Y 256.133,Z 211.74,A -85,B 0,C 180,E1 -18394.722,E2 -18394.722} C_VEL
LIN {X 0,Y 257.576,Z 217.612,A -85,B 0,C 180,E1 -18398.87,E2 -18398.87} C_VEL
LIN {X 0,Y 259.076,Z 224.043,A -85,B 0,C 180,E1 -18402.913,E2 -18402.913} C_VEL
LIN {X 0,Y 260.584,Z 230.736,A -85,B 0,C 180,E1 -18406.735,E2 -18406.735} C_VEL
LIN {X 0,Y 262.233,Z 238.064,A -85,B 0,C 180,E1 -18410.564,E2 -18410.564} C_VEL
LIN {X 0,Y 263.742,Z 245.283,A -85,B 0,C 180,E1 -18414.112,E2 -18414.112} C_VEL
LIN {X 0,Y 264.281,Z 248.334,A -85,B 0,C 180,E1 -18415.526,E2 -18415.526} C_VEL
LIN {X 0,Y 263.914,Z 250.533,A -85,B 0,C 180,E1 -18416.459,E2 -18416.459} C_VEL
LIN {X 0,Y 260.123,Z 263.496,A -85,B 0,C 180,E1 -18421.785,E2 -18421.785} C_VEL
LIN {X 0,Y 258.397,Z 270.574,A -85,B 0,C 180,E1 -18424.719,E2 -18424.719} C_VEL
LIN {X 0,Y 259.629,Z 283.3,A -85,B 0,C 180,E1 -18425.515,E2 -18425.515} C_VEL
LIN {X 0,Y 260.087,Z 295.705,A -85,B 0,C 180,E1 -18426.583,E2 -18426.583} C_VEL
LIN {X 0,Y 259.964,Z 306.434,A -85,B 0,C 180,E1 -18427.763,E2 -18427.763} C_VEL
LIN {X 0,Y 259.916,Z 316.776,A -85,B 0,C 180,E1 -18429.215,E2 -18429.215} C_VEL
LIN {X 0,Y 259.476,Z 324.168,A -85,B 0,C 180,E1 -18430.419,E2 -18430.419} C_VEL
LIN {X 0,Y 258.064,Z 333.18,A -85,B 0,C 180,E1 -18432.161,E2 -18432.161} C_VEL
LIN {X 0,Y 257.143,Z 340.091,A -85,B 0,C 180,E1 -18433.759,E2 -18433.759} C_VEL
LIN {X 0,Y 256.393,Z 346,A -85,B 0,C 180,E1 -18435.314,E2 -18435.314} C_VEL
LIN {X 0,Y 255.639,Z 355.077,A -85,B 0,C 180,E1 -18437.297,E2 -18437.297} C_VEL
LIN {X 0,Y 255.109,Z 362.642,A -85,B 0,C 180,E1 -18439.285,E2 -18439.285} C_VEL
LIN {X 0,Y 254.835,Z 370.091,A -85,B 0,C 180,E1 -18441.677,E2 -18441.677} C_VEL
LIN {X 0,Y 254.73,Z 376.868,A -85,B 0,C 180,E1 -18444.461,E2 -18444.461} C_VEL
LIN {X 0,Y 254.769,Z 381.297,A -85,B 0,C 180,E1 -18446.839,E2 -18446.839} C_VEL
LIN {X 0,Y 254.81,Z 383.595,A -85,B 0,C 180,E1 -18448.422,E2 -18448.422} C_VEL
LIN {X 0,Y 254.813,Z 385.389,A -85,B 0,C 180,E1 -18450.002,E2 -18450.002} C_VEL
LIN {X 0,Y 254.641,Z 386.735,A -85,B 0,C 180,E1 -18451.584,E2 -18451.584} C_VEL
LIN {X 0,Y 254.295,Z 387.65,A -85,B 0,C 180,E1 -18453.171,E2 -18453.171} C_VEL
LIN {X 0,Y 254.228,Z 388.276,A -85,B 0,C 180,E1 -18455.615,E2 -18455.615} C_VEL
LIN {X 0,Y 254.349,Z 388.02,A -85,B 0,C 180,E1 -18457.943,E2 -18457.943} C_VEL
LIN {X 0,Y 255.179,Z 386.416,A -85,B 0,C 180,E1 -18461.118,E2 -18461.118} C_VEL
LIN {X 0,Y 256.768,Z 383.301,A -85,B 0,C 180,E1 -18464.263,E2 -18464.263} C_VEL
LIN {X 0,Y 259.517,Z 378.698,A -85,B 0,C 180,E1 -18467.333,E2 -18467.333} C_VEL
LIN {X 0,Y 262.79,Z 372.498,A -85,B 0,C 180,E1 -18470.347,E2 -18470.347} C_VEL
LIN {X 0,Y 265.972,Z 366.698,A -85,B 0,C 180,E1 -18472.531,E2 -18472.531} C_VEL
LIN {X 0,Y 270.499,Z 358.505,A -85,B 0,C 180,E1 -18474.975,E2 -18474.975} C_VEL
LIN {X 0,Y 275.688,Z 348.544,A -85,B 0,C 180,E1 -18477.316,E2 -18477.316} C_VEL
LIN {X 0,Y 280.587,Z 338.346,A -85,B 0,C 180,E1 -18479.239,E2 -18479.239} C_VEL
LIN {X 0,Y 284.984,Z 326.765,A -85,B 0,C 180,E1 -18481.192,E2 -18481.192} C_VEL
LIN {X 0,Y 287.749,Z 316.692,A -85,B 0,C 180,E1 -18482.871,E2 -18482.871} C_VEL
LIN {X 0,Y 289.563,Z 306.669,A -85,B 0,C 180,E1 -18484.659,E2 -18484.659} C_VEL
LIN {X 0,Y 290.796,Z 296.458,A -85,B 0,C 180,E1 -18486.624,E2 -18486.624} C_VEL
LIN {X 0,Y 291.226,Z 290.226,A -85,B 0,C 180,E1 -18488,E2 -18488} C_VEL
LIN {X 0,Y 291.173,Z 288.716,A -85,B 0,C 180,E1 -18488.439,E2 -18488.439} C_VEL
LIN {X 0,Y 290.77,Z 286.616,A -85,B 0,C 180,E1 -18489.335,E2 -18489.335} C_VEL
LIN {X 0,Y 289.883,Z 284.222,A -85,B 0,C 180,E1 -18490.891,E2 -18490.891} C_VEL
LIN {X 0,Y 288.775,Z 282.544,A -85,B 0,C 180,E1 -18493.103,E2 -18493.103} C_VEL
LIN {X 0,Y 288.131,Z 282.344,A -85,B 0,C 180,E1 -18495.022,E2 -18495.022} C_VEL
LIN {X 0,Y 287.9,Z 283.01,A -85,B 0,C 180,E1 -18497.085,E2 -18497.085} C_VEL
LIN {X 0,Y 288.007,Z 284.766,A -85,B 0,C 180,E1 -18499.156,E2 -18499.156} C_VEL
LIN {X 0,Y 288.226,Z 286.827,A -85,B 0,C 180,E1 -18500.656,E2 -18500.656} C_VEL
LIN {X 0,Y 288.26,Z 291.938,A -85,B 0,C 180,E1 -18502.911,E2 -18502.911} C_VEL
LIN {X 0,Y 288.456,Z 299.09,A -85,B 0,C 180,E1 -18505.54,E2 -18505.54} C_VEL
LIN {X 0,Y 288.438,Z 307.488,A -85,B 0,C 180,E1 -18508.197,E2 -18508.197} C_VEL
LIN {X 0,Y 287.82,Z 314.459,A -85,B 0,C 180,E1 -18510.115,E2 -18510.115} C_VEL
LIN {X 0,Y 285.769,Z 319.223,A -85,B 0,C 180,E1 -18510.94,E2 -18510.94} C_VEL
LIN {X 0,Y 280.889,Z 329.084,A -85,B 0,C 180,E1 -18512.83,E2 -18512.83} C_VEL
LIN {X 0,Y 275.735,Z 338.516,A -85,B 0,C 180,E1 -18515.13,E2 -18515.13} C_VEL
LIN {X 0,Y 271.702,Z 345.185,A -85,B 0,C 180,E1 -18517.17,E2 -18517.17} C_VEL
LIN {X 0,Y 268.125,Z 350.696,A -85,B 0,C 180,E1 -18519.277,E2 -18519.277} C_VEL
LIN {X 0,Y 264.984,Z 355.172,A -85,B 0,C 180,E1 -18521.442,E2 -18521.442} C_VEL
LIN {X 0,Y 261.588,Z 359.662,A -85,B 0,C 180,E1 -18524.415,E2 -18524.415} C_VEL
LIN {X 0,Y 258.787,Z 362.592,A -85,B 0,C 180,E1 -18527.452,E2 -18527.452} C_VEL
LIN {X 0,Y 257.792,Z 363.498,A -85,B 0,C 180,E1 -18528.998,E2 -18528.998} C_VEL
LIN {X 0,Y 256.631,Z 364.072,A -85,B 0,C 180,E1 -18530.543,E2 -18530.543} C_VEL
LIN {X 0,Y 255.431,Z 363.999,A -85,B 0,C 180,E1 -18533.681,E2 -18533.681} C_VEL
LIN {X 0,Y 254.626,Z 362.472,A -85,B 0,C 180,E1 -18536.836,E2 -18536.836} C_VEL
LIN {X 0,Y 254.233,Z 359.331,A -85,B 0,C 180,E1 -18540,E2 -18540} C_VEL
LIN {X 0,Y 254.274,Z 355.899,A -85,B 0,C 180,E1 -18542.376,E2 -18542.376} C_VEL
LIN {X 0,Y 254.345,Z 351.422,A -85,B 0,C 180,E1 -18544.755,E2 -18544.755} C_VEL
LIN {X 0,Y 254.723,Z 344.762,A -85,B 0,C 180,E1 -18547.531,E2 -18547.531} C_VEL
LIN {X 0,Y 255.365,Z 336.194,A -85,B 0,C 180,E1 -18550.305,E2 -18550.305} C_VEL
LIN {X 0,Y 256.175,Z 327.08,A -85,B 0,C 180,E1 -18552.678,E2 -18552.678} C_VEL
LIN {X 0,Y 257.345,Z 315.852,A -85,B 0,C 180,E1 -18555.037,E2 -18555.037} C_VEL
LIN {X 0,Y 258.487,Z 304.22,A -85,B 0,C 180,E1 -18556.995,E2 -18556.995} C_VEL
LIN {X 0,Y 259.488,Z 292.793,A -85,B 0,C 180,E1 -18558.564,E2 -18558.564} C_VEL
LIN {X 0,Y 260.299,Z 282.404,A -85,B 0,C 180,E1 -18559.725,E2 -18559.725} C_VEL
LIN {X 0,Y 258.197,Z 268.551,A -85,B 0,C 180,E1 -18561.025,E2 -18561.025} C_VEL
LIN {X 0,Y 256.414,Z 254.469,A -85,B 0,C 180,E1 -18562.013,E2 -18562.013} C_VEL
LIN {X 0,Y 256.379,Z 253.689,A -85,B 0,C 180,E1 -18562.095,E2 -18562.095} C_VEL
LIN {X 0,Y 256.856,Z 245.796,A -85,B 0,C 180,E1 -18565.963,E2 -18565.963} C_VEL
LIN {X 0,Y 257.427,Z 236.955,A -85,B 0,C 180,E1 -18570.336,E2 -18570.336} C_VEL
LIN {X 0,Y 257.95,Z 229.695,A -85,B 0,C 180,E1 -18573.955,E2 -18573.955} C_VEL
LIN {X 0,Y 258.2,Z 224.07,A -85,B 0,C 180,E1 -18576.786,E2 -18576.786} C_VEL
LIN {X 0,Y 257.289,Z 217.761,A -85,B 0,C 180,E1 -18580.105,E2 -18580.105} C_VEL
LIN {X 0,Y 256.108,Z 211.584,A -85,B 0,C 180,E1 -18583.436,E2 -18583.436} C_VEL
LIN {X 0,Y 256.078,Z 211.586,A -85,B 0,C 180,E1 -18587.818,E2 -18587.818} C_VEL
LIN {X 0,Y 256.154,Z 211.802,A -85,B 0,C 180,E1 -18591.864,E2 -18591.864} C_VEL
LIN {X 0,Y 256.658,Z 214.612,A -85,B 0,C 180,E1 -18595.234,E2 -18595.234} C_VEL
LIN {X 0,Y 257.003,Z 217.69,A -85,B 0,C 180,E1 -18598.694,E2 -18598.694} C_VEL
LIN {X 0,Y 257.008,Z 221.134,A -85,B 0,C 180,E1 -18602.296,E2 -18602.296} C_VEL
LIN {X 0,Y 256.877,Z 224.699,A -85,B 0,C 180,E1 -18605.769,E2 -18605.769} C_VEL
LIN {X 0,Y 256.717,Z 229.407,A -85,B 0,C 180,E1 -18609.999,E2 -18609.999} C_VEL
LIN {X 0,Y 260.141,Z 240.248,A -85,B 0,C 180,E1 -18611.009,E2 -18611.009} C_VEL
LIN {X 0,Y 262.456,Z 249.657,A -85,B 0,C 180,E1 -18612.123,E2 -18612.123} C_VEL
LIN {X 0,Y 264.003,Z 258.537,A -85,B 0,C 180,E1 -18613.407,E2 -18613.407} C_VEL
LIN {X 0,Y 263.07,Z 266.637,A -85,B 0,C 180,E1 -18614.702,E2 -18614.702} C_VEL
LIN {X 0,Y 262.061,Z 273.268,A -85,B 0,C 180,E1 -18616.031,E2 -18616.031} C_VEL
LIN {X 0,Y 260.824,Z 279.465,A -85,B 0,C 180,E1 -18617.55,E2 -18617.55} C_VEL
LIN {X 0,Y 259.742,Z 284.352,A -85,B 0,C 180,E1 -18619.08,E2 -18619.08} C_VEL
LIN {X 0,Y 258.812,Z 288.289,A -85,B 0,C 180,E1 -18620.621,E2 -18620.621} C_VEL
LIN {X 0,Y 258.172,Z 292.673,A -85,B 0,C 180,E1 -18622.962,E2 -18622.962} C_VEL
LIN {X 0,Y 257.219,Z 295.654,A -85,B 0,C 180,E1 -18625.296,E2 -18625.296} C_VEL
LIN {X 0,Y 256.994,Z 296.906,A -85,B 0,C 180,E1 -18626.863,E2 -18626.863} C_VEL
LIN {X 0,Y 256.76,Z 297.67,A -85,B 0,C 180,E1 -18628.43,E2 -18628.43} C_VEL
LIN {X 0,Y 256.668,Z 297.939,A -85,B 0,C 180,E1 -18629.998,E2 -18629.998} C_VEL
LIN {X 0,Y 256.758,Z 297.705,A -85,B 0,C 180,E1 -18631.566,E2 -18631.566} C_VEL
LIN {X 0,Y 256.991,Z 296.989,A -85,B 0,C 180,E1 -18633.133,E2 -18633.133} C_VEL
LIN {X 0,Y 257.216,Z 295.788,A -85,B 0,C 180,E1 -18634.7,E2 -18634.7} C_VEL
LIN {X 0,Y 258.161,Z 292.866,A -85,B 0,C 180,E1 -18637.035,E2 -18637.035} C_VEL
LIN {X 0,Y 258.773,Z 288.57,A -85,B 0,C 180,E1 -18639.376,E2 -18639.376} C_VEL
LIN {X 0,Y 259.566,Z 285.746,A -85,B 0,C 180,E1 -18640.529,E2 -18640.529} C_VEL
LIN {X 0,Y 260.503,Z 281.2,A -85,B 0,C 180,E1 -18642.067,E2 -18642.067} C_VEL
LIN {X 0,Y 261.726,Z 275.489,A -85,B 0,C 180,E1 -18643.587,E2 -18643.587} C_VEL
LIN {X 0,Y 262.863,Z 268.324,A -85,B 0,C 180,E1 -18645.108,E2 -18645.108} C_VEL
LIN {X 0,Y 263.629,Z 261.922,A -85,B 0,C 180,E1 -18646.207,E2 -18646.207} C_VEL
LIN {X 0,Y 263.92,Z 257.487,A -85,B 0,C 180,E1 -18646.879,E2 -18646.879} C_VEL
LIN {X 0,Y 262.161,Z 247.865,A -85,B 0,C 180,E1 -18648.232,E2 -18648.232} C_VEL
LIN {X 0,Y 259.168,Z 236.985,A -85,B 0,C 180,E1 -18649.456,E2 -18649.456} C_VEL
LIN {X 0,Y 256.718,Z 229.318,A -85,B 0,C 180,E1 -18650.139,E2 -18650.139} C_VEL
LIN {X 0,Y 256.882,Z 224.853,A -85,B 0,C 180,E1 -18654.226,E2 -18654.226} C_VEL
LIN {X 0,Y 257.008,Z 221.337,A -85,B 0,C 180,E1 -18657.699,E2 -18657.699} C_VEL
LIN {X 0,Y 257.009,Z 217.89,A -85,B 0,C 180,E1 -18661.3,E2 -18661.3} C_VEL
LIN {X 0,Y 256.609,Z 214.472,A -85,B 0,C 180,E1 -18665.107,E2 -18665.107} C_VEL
LIN {X 0,Y 256.102,Z 211.586,A -85,B 0,C 180,E1 -18668.642,E2 -18668.642} C_VEL
LIN {X 0,Y 256.059,Z 211.587,A -85,B 0,C 180,E1 -18673.324,E2 -18673.324} C_VEL
LIN {X 0,Y 256.081,Z 211.588,A -85,B 0,C 180,E1 -18677.813,E2 -18677.813} C_VEL
LIN {X 0,Y 256.084,Z 211.588,A -85,B 0,C 180,E1 -18680.86,E2 -18680.86} C_VEL
LIN {X 0,Y 256.101,Z 211.584,A -85,B 0,C 180,E1 -18684.81,E2 -18684.81} C_VEL
LIN {X 0,Y 256.085,Z 211.587,A -85,B 0,C 180,E1 -18688.571,E2 -18688.571} C_VEL
LIN {X 0,Y 256.133,Z 211.579,A -85,B 0,C 180,E1 -18692.195,E2 -18692.195} C_VEL
LIN {X 0,Y 256.158,Z 211.566,A -85,B 0,C 180,E1 -18695.698,E2 -18695.698} C_VEL
LIN {X 0,Y 256.157,Z 211.566,A -85,B 0,C 180,E1 -18699.104,E2 -18699.104} C_VEL
LIN {X 0,Y 256.29,Z 211.548,A -85,B 0,C 180,E1 -18704.084,E2 -18704.084} C_VEL
LIN {X 0,Y 256.285,Z 211.562,A -85,B 0,C 180,E1 -18707.327,E2 -18707.327} C_VEL
LIN {X 0,Y 256.505,Z 211.532,A -85,B 0,C 180,E1 -18712.126,E2 -18712.126} C_VEL
LIN {X 0,Y 256.488,Z 211.531,A -85,B 0,C 180,E1 -18716.858,E2 -18716.858} C_VEL
LIN {X 0,Y 256.754,Z 211.487,A -85,B 0,C 180,E1 -18720,E2 -18720} C_VEL
LIN {X 0,Y 256.485,Z 211.533,A -85,B 0,C 180,E1 -18723.141,E2 -18723.141} C_VEL
LIN {X 0,Y 256.529,Z 211.529,A -85,B 0,C 180,E1 -18727.873,E2 -18727.873} C_VEL
LIN {X 0,Y 256.298,Z 211.56,A -85,B 0,C 180,E1 -18731.066,E2 -18731.066} C_VEL
LIN {X 0,Y 256.221,Z 211.561,A -85,B 0,C 180,E1 -18734.292,E2 -18734.292} C_VEL
LIN {X 0,Y 256.117,Z 211.574,A -85,B 0,C 180,E1 -18738.119,E2 -18738.119} C_VEL
LIN {X 0,Y 256.109,Z 211.585,A -85,B 0,C 180,E1 -18741.098,E2 -18741.098} C_VEL
LIN {X 0,Y 256.072,Z 211.59,A -85,B 0,C 180,E1 -18744.944,E2 -18744.944} C_VEL
LIN {X 0,Y 255.41,Z 211.676,A -85,B 0,C 180,E1 -18746.256,E2 -18746.256} C_VEL
LIN {X 0,Y 252.509,Z 212.035,A -85,B 0,C 180,E1 -18748.395,E2 -18748.395} C_VEL
LIN {X 0,Y 250.066,Z 212.338,A -85,B 0,C 180,E1 -18750.136,E2 -18750.136} C_VEL
LIN {X 0,Y 249.064,Z 212.462,A -85,B 0,C 180,E1 -18751.487,E2 -18751.487} C_VEL
LIN {X 0,Y 249.009,Z 212.466,A -85,B 0,C 180,E1 -18751.945,E2 -18751.945} C_VEL
LIN {X 0,Y 249.031,Z 212.614,A -85,B 0,C 180,E1 -18753.389,E2 -18753.389} C_VEL
LIN {X 0,Y 250.313,Z 217.562,A -85,B 0,C 180,E1 -18757.132,E2 -18757.132} C_VEL
LIN {X 0,Y 251.67,Z 223.339,A -85,B 0,C 180,E1 -18761.067,E2 -18761.067} C_VEL
LIN {X 0,Y 253.136,Z 229.878,A -85,B 0,C 180,E1 -18765.07,E2 -18765.07} C_VEL
LIN {X 0,Y 254.873,Z 237.569,A -85,B 0,C 180,E1 -18769.337,E2 -18769.337} C_VEL
LIN {X 0,Y 256.539,Z 245.56,A -85,B 0,C 180,E1 -18773.43,E2 -18773.43} C_VEL
LIN {X 0,Y 257.188,Z 248.913,A -85,B 0,C 180,E1 -18775.064,E2 -18775.064} C_VEL
LIN {X 0,Y 257.138,Z 250.905,A -85,B 0,C 180,E1 -18775.966,E2 -18775.966} C_VEL
LIN {X 0,Y 252.959,Z 264.647,A -85,B 0,C 180,E1 -18781.818,E2 -18781.818} C_VEL
LIN {X 0,Y 251.64,Z 269.864,A -85,B 0,C 180,E1 -18784.073,E2 -18784.073} C_VEL
LIN {X 0,Y 252.817,Z 282.591,A -85,B 0,C 180,E1 -18784.892,E2 -18784.892} C_VEL
LIN {X 0,Y 253.302,Z 294.133,A -85,B 0,C 180,E1 -18785.912,E2 -18785.912} C_VEL
LIN {X 0,Y 253.158,Z 305.091,A -85,B 0,C 180,E1 -18787.131,E2 -18787.131} C_VEL
LIN {X 0,Y 253.055,Z 315.575,A -85,B 0,C 180,E1 -18788.625,E2 -18788.625} C_VEL
LIN {X 0,Y 252.558,Z 324.092,A -85,B 0,C 180,E1 -18790.072,E2 -18790.072} C_VEL
LIN {X 0,Y 251.233,Z 332.099,A -85,B 0,C 180,E1 -18791.659,E2 -18791.659} C_VEL
LIN {X 0,Y 250.058,Z 340.408,A -85,B 0,C 180,E1 -18793.679,E2 -18793.679} C_VEL
LIN {X 0,Y 249.096,Z 348.332,A -85,B 0,C 180,E1 -18795.918,E2 -18795.918} C_VEL
LIN {X 0,Y 248.376,Z 357.66,A -85,B 0,C 180,E1 -18798.164,E2 -18798.164} C_VEL
LIN {X 0,Y 247.893,Z 365.976,A -85,B 0,C 180,E1 -18800.62,E2 -18800.62} C_VEL
LIN {X 0,Y 247.723,Z 372.919,A -85,B 0,C 180,E1 -18803.201,E2 -18803.201} C_VEL
LIN {X 0,Y 247.686,Z 378.631,A -85,B 0,C 180,E1 -18805.934,E2 -18805.934} C_VEL
LIN {X 0,Y 247.798,Z 382.478,A -85,B 0,C 180,E1 -18808.377,E2 -18808.377} C_VEL
LIN {X 0,Y 247.792,Z 384.424,A -85,B 0,C 180,E1 -18810.002,E2 -18810.002} C_VEL
LIN {X 0,Y 247.595,Z 385.854,A -85,B 0,C 180,E1 -18811.629,E2 -18811.629} C_VEL
LIN {X 0,Y 247.199,Z 387.508,A -85,B 0,C 180,E1 -18814.895,E2 -18814.895} C_VEL
LIN {X 0,Y 247.313,Z 387.633,A -85,B 0,C 180,E1 -18818.171,E2 -18818.171} C_VEL
LIN {X 0,Y 248.186,Z 386.255,A -85,B 0,C 180,E1 -18821.435,E2 -18821.435} C_VEL
LIN {X 0,Y 249.893,Z 383.468,A -85,B 0,C 180,E1 -18824.664,E2 -18824.664} C_VEL
LIN {X 0,Y 252.77,Z 379.178,A -85,B 0,C 180,E1 -18827.811,E2 -18827.811} C_VEL
LIN {X 0,Y 256.209,Z 373.379,A -85,B 0,C 180,E1 -18830.893,E2 -18830.893} C_VEL
LIN {X 0,Y 260.179,Z 366.919,A -85,B 0,C 180,E1 -18833.482,E2 -18833.482} C_VEL
LIN {X 0,Y 264.967,Z 358.951,A -85,B 0,C 180,E1 -18835.956,E2 -18835.956} C_VEL
LIN {X 0,Y 270.425,Z 349.355,A -85,B 0,C 180,E1 -18838.315,E2 -18838.315} C_VEL
LIN {X 0,Y 276.365,Z 337.747,A -85,B 0,C 180,E1 -18840.573,E2 -18840.573} C_VEL
LIN {X 0,Y 280.215,Z 328.462,A -85,B 0,C 180,E1 -18842.208,E2 -18842.208} C_VEL
LIN {X 0,Y 283.195,Z 319.154,A -85,B 0,C 180,E1 -18843.847,E2 -18843.847} C_VEL
LIN {X 0,Y 285.633,Z 308.357,A -85,B 0,C 180,E1 -18845.897,E2 -18845.897} C_VEL
LIN {X 0,Y 287.098,Z 299.527,A -85,B 0,C 180,E1 -18847.735,E2 -18847.735} C_VEL
LIN {X 0,Y 287.734,Z 294.418,A -85,B 0,C 180,E1 -18848.958,E2 -18848.958} C_VEL
LIN {X 0,Y 287.444,Z 292.279,A -85,B 0,C 180,E1 -18849.928,E2 -18849.928} C_VEL
LIN {X 0,Y 287.15,Z 291.109,A -85,B 0,C 180,E1 -18850.648,E2 -18850.648} C_VEL
LIN {X 0,Y 286.188,Z 289.438,A -85,B 0,C 180,E1 -18852.547,E2 -18852.547} C_VEL
LIN {X 0,Y 285.461,Z 288.877,A -85,B 0,C 180,E1 -18854.441,E2 -18854.441} C_VEL
LIN {X 0,Y 285.013,Z 289.255,A -85,B 0,C 180,E1 -18856.335,E2 -18856.335} C_VEL
LIN {X 0,Y 284.9,Z 290.41,A -85,B 0,C 180,E1 -18858.237,E2 -18858.237} C_VEL
LIN {X 0,Y 284.926,Z 292.594,A -85,B 0,C 180,E1 -18860.11,E2 -18860.11} C_VEL
LIN {X 0,Y 284.613,Z 296.943,A -85,B 0,C 180,E1 -18862.205,E2 -18862.205} C_VEL
LIN {X 0,Y 284.301,Z 303.185,A -85,B 0,C 180,E1 -18864.666,E2 -18864.666} C_VEL
LIN {X 0,Y 283.782,Z 311.064,A -85,B 0,C 180,E1 -18867.357,E2 -18867.357} C_VEL
LIN {X 0,Y 282.817,Z 317.645,A -85,B 0,C 180,E1 -18869.314,E2 -18869.314} C_VEL
LIN {X 0,Y 277.549,Z 327.952,A -85,B 0,C 180,E1 -18871.242,E2 -18871.242} C_VEL
LIN {X 0,Y 271.915,Z 337.66,A -85,B 0,C 180,E1 -18873.522,E2 -18873.522} C_VEL
LIN {X 0,Y 266.812,Z 345.514,A -85,B 0,C 180,E1 -18875.903,E2 -18875.903} C_VEL
LIN {X 0,Y 262.915,Z 351.025,A -85,B 0,C 180,E1 -18878.023,E2 -18878.023} C_VEL
LIN {X 0,Y 258.457,Z 356.809,A -85,B 0,C 180,E1 -18880.955,E2 -18880.955} C_VEL
LIN {X 0,Y 254.87,Z 360.904,A -85,B 0,C 180,E1 -18883.993,E2 -18883.993} C_VEL
LIN {X 0,Y 251.934,Z 363.548,A -85,B 0,C 180,E1 -18887.105,E2 -18887.105} C_VEL
LIN {X 0,Y 250.877,Z 364.276,A -85,B 0,C 180,E1 -18888.691,E2 -18888.691} C_VEL
LIN {X 0,Y 249.662,Z 364.69,A -85,B 0,C 180,E1 -18890.276,E2 -18890.276} C_VEL
LIN {X 0,Y 248.402,Z 364.379,A -85,B 0,C 180,E1 -18893.502,E2 -18893.502} C_VEL
LIN {X 0,Y 247.959,Z 363.65,A -85,B 0,C 180,E1 -18895.122,E2 -18895.122} C_VEL
LIN {X 0,Y 247.299,Z 361.051,A -85,B 0,C 180,E1 -18898.372,E2 -18898.372} C_VEL
LIN {X 0,Y 247.134,Z 358.057,A -85,B 0,C 180,E1 -18900.815,E2 -18900.815} C_VEL
LIN {X 0,Y 247.239,Z 354.083,A -85,B 0,C 180,E1 -18903.259,E2 -18903.259} C_VEL
LIN {X 0,Y 247.361,Z 348.249,A -85,B 0,C 180,E1 -18906.043,E2 -18906.043} C_VEL
LIN {X 0,Y 247.82,Z 341.544,A -85,B 0,C 180,E1 -18908.562,E2 -18908.562} C_VEL
LIN {X 0,Y 248.476,Z 333.553,A -85,B 0,C 180,E1 -18911.007,E2 -18911.007} C_VEL
LIN {X 0,Y 249.209,Z 325.53,A -85,B 0,C 180,E1 -18913.039,E2 -18913.039} C_VEL
LIN {X 0,Y 250.344,Z 314.926,A -85,B 0,C 180,E1 -18915.259,E2 -18915.259} C_VEL
LIN {X 0,Y 251.501,Z 303.104,A -85,B 0,C 180,E1 -18917.272,E2 -18917.272} C_VEL
LIN {X 0,Y 252.627,Z 290.883,A -85,B 0,C 180,E1 -18918.934,E2 -18918.934} C_VEL
LIN {X 0,Y 253.163,Z 282.499,A -85,B 0,C 180,E1 -18919.881,E2 -18919.881} C_VEL
LIN {X 0,Y 251.045,Z 268.476,A -85,B 0,C 180,E1 -18921.235,E2 -18921.235} C_VEL
LIN {X 0,Y 249.329,Z 254.045,A -85,B 0,C 180,E1 -18922.293,E2 -18922.293} C_VEL
LIN {X 0,Y 249.9,Z 245.121,A -85,B 0,C 180,E1 -18926.742,E2 -18926.742} C_VEL
LIN {X 0,Y 250.52,Z 236.128,A -85,B 0,C 180,E1 -18931.265,E2 -18931.265} C_VEL
LIN {X 0,Y 251.092,Z 228.949,A -85,B 0,C 180,E1 -18934.906,E2 -18934.906} C_VEL
LIN {X 0,Y 251.177,Z 224.91,A -85,B 0,C 180,E1 -18936.983,E2 -18936.983} C_VEL
LIN {X 0,Y 250.272,Z 218.862,A -85,B 0,C 180,E1 -18940.231,E2 -18940.231} C_VEL
LIN {X 0,Y 249.078,Z 212.46,A -85,B 0,C 180,E1 -18943.788,E2 -18943.788} C_VEL
LIN {X 0,Y 249.022,Z 212.464,A -85,B 0,C 180,E1 -18947.362,E2 -18947.362} C_VEL
LIN {X 0,Y 249.073,Z 212.672,A -85,B 0,C 180,E1 -18950.848,E2 -18950.848} C_VEL
LIN {X 0,Y 249.653,Z 215.777,A -85,B 0,C 180,E1 -18954.725,E2 -18954.725} C_VEL
LIN {X 0,Y 250.014,Z 218.35,A -85,B 0,C 180,E1 -18957.715,E2 -18957.715} C_VEL
LIN {X 0,Y 250.099,Z 221.826,A -85,B 0,C 180,E1 -18961.462,E2 -18961.462} C_VEL
LIN {X 0,Y 249.946,Z 225.399,A -85,B 0,C 180,E1 -18965.052,E2 -18965.052} C_VEL
LIN {X 0,Y 249.807,Z 230.165,A -85,B 0,C 180,E1 -18969.339,E2 -18969.339} C_VEL
LIN {X 0,Y 253.05,Z 240.358,A -85,B 0,C 180,E1 -18970.325,E2 -18970.325} C_VEL
LIN {X 0,Y 255.316,Z 249.003,A -85,B 0,C 180,E1 -18971.362,E2 -18971.362} C_VEL
LIN {X 0,Y 257.184,Z 258.623,A -85,B 0,C 180,E1 -18972.782,E2 -18972.782} C_VEL
LIN {X 0,Y 256.677,Z 265.065,A -85,B 0,C 180,E1 -18973.799,E2 -18973.799} C_VEL
LIN {X 0,Y 255.558,Z 272.658,A -85,B 0,C 180,E1 -18975.261,E2 -18975.261} C_VEL
LIN {X 0,Y 254.271,Z 279.079,A -85,B 0,C 180,E1 -18976.817,E2 -18976.817} C_VEL
LIN {X 0,Y 252.845,Z 285.353,A -85,B 0,C 180,E1 -18978.778,E2 -18978.778} C_VEL
LIN {X 0,Y 251.879,Z 289.278,A -85,B 0,C 180,E1 -18980.361,E2 -18980.361} C_VEL
LIN {X 0,Y 251.199,Z 293.653,A -85,B 0,C 180,E1 -18982.765,E2 -18982.765} C_VEL
LIN {X 0,Y 250.216,Z 296.63,A -85,B 0,C 180,E1 -18985.164,E2 -18985.164} C_VEL
LIN {X 0,Y 249.978,Z 297.88,A -85,B 0,C 180,E1 -18986.775,E2 -18986.775} C_VEL
LIN {X 0,Y 249.735,Z 298.643,A -85,B 0,C 180,E1 -18988.385,E2 -18988.385} C_VEL
LIN {X 0,Y 249.64,Z 298.914,A -85,B 0,C 180,E1 -18989.998,E2 -18989.998} C_VEL
LIN {X 0,Y 249.734,Z 298.678,A -85,B 0,C 180,E1 -18991.611,E2 -18991.611} C_VEL
LIN {X 0,Y 249.975,Z 297.963,A -85,B 0,C 180,E1 -18993.221,E2 -18993.221} C_VEL
LIN {X 0,Y 250.213,Z 296.763,A -85,B 0,C 180,E1 -18994.832,E2 -18994.832} C_VEL
LIN {X 0,Y 251.187,Z 293.842,A -85,B 0,C 180,E1 -18997.231,E2 -18997.231} C_VEL
LIN {X 0,Y 251.839,Z 289.556,A -85,B 0,C 180,E1 -18999.637,E2 -18999.637} C_VEL
LIN {X 0,Y 252.529,Z 287.702,A -85,B 0,C 180,E1 -19000.42,E2 -19000.42} C_VEL
LIN {X 0,Y 253.322,Z 283.439,A -85,B 0,C 180,E1 -19002.007,E2 -19002.007} C_VEL
LIN {X 0,Y 254.911,Z 276.541,A -85,B 0,C 180,E1 -19003.958,E2 -19003.958} C_VEL
LIN {X 0,Y 256.098,Z 269.419,A -85,B 0,C 180,E1 -19005.517,E2 -19005.517} C_VEL
LIN {X 0,Y 256.928,Z 262.883,A -85,B 0,C 180,E1 -19006.675,E2 -19006.675} C_VEL
LIN {X 0,Y 257.312,Z 259.917,A -85,B 0,C 180,E1 -19007.137,E2 -19007.137} C_VEL
LIN {X 0,Y 255.863,Z 251.198,A -85,B 0,C 180,E1 -19008.463,E2 -19008.463} C_VEL
LIN {X 0,Y 253.368,Z 241.217,A -85,B 0,C 180,E1 -19009.709,E2 -19009.709} C_VEL
LIN {X 0,Y 249.77,Z 229.93,A -85,B 0,C 180,E1 -19010.851,E2 -19010.851} C_VEL
LIN {X 0,Y 250.016,Z 224.593,A -85,B 0,C 180,E1 -19015.904,E2 -19015.904} C_VEL
LIN {X 0,Y 250.101,Z 221.15,A -85,B 0,C 180,E1 -19019.41,E2 -19019.41} C_VEL
LIN {X 0,Y 249.995,Z 218.329,A -85,B 0,C 180,E1 -19022.501,E2 -19022.501} C_VEL
LIN {X 0,Y 249.525,Z 215.102,A -85,B 0,C 180,E1 -19026.259,E2 -19026.259} C_VEL
LIN {X 0,Y 249.022,Z 212.464,A -85,B 0,C 180,E1 -19029.679,E2 -19029.679} C_VEL
LIN {X 0,Y 249.006,Z 212.47,A -85,B 0,C 180,E1 -19032.791,E2 -19032.791} C_VEL
LIN {X 0,Y 249.022,Z 212.465,A -85,B 0,C 180,E1 -19037.364,E2 -19037.364} C_VEL
LIN {X 0,Y 249.029,Z 212.463,A -85,B 0,C 180,E1 -19041.62,E2 -19041.62} C_VEL
LIN {X 0,Y 249.048,Z 212.456,A -85,B 0,C 180,E1 -19045.64,E2 -19045.64} C_VEL
LIN {X 0,Y 249.044,Z 212.458,A -85,B 0,C 180,E1 -19049.472,E2 -19049.472} C_VEL
LIN {X 0,Y 249.065,Z 212.46,A -85,B 0,C 180,E1 -19053.161,E2 -19053.161} C_VEL
LIN {X 0,Y 249.07,Z 212.46,A -85,B 0,C 180,E1 -19056.732,E2 -19056.732} C_VEL
LIN {X 0,Y 249.101,Z 212.444,A -85,B 0,C 180,E1 -19060.211,E2 -19060.211} C_VEL
LIN {X 0,Y 249.232,Z 212.431,A -85,B 0,C 180,E1 -19063.621,E2 -19063.621} C_VEL
LIN {X 0,Y 249.235,Z 212.433,A -85,B 0,C 180,E1 -19068.616,E2 -19068.616} C_VEL
LIN {X 0,Y 249.444,Z 212.411,A -85,B 0,C 180,E1 -19071.902,E2 -19071.902} C_VEL
LIN {X 0,Y 249.285,Z 212.418,A -85,B 0,C 180,E1 -19075.148,E2 -19075.148} C_VEL
LIN {X 0,Y 249.665,Z 212.382,A -85,B 0,C 180,E1 -19078.387,E2 -19078.387} C_VEL
LIN {X 0,Y 249.664,Z 212.382,A -85,B 0,C 180,E1 -19081.613,E2 -19081.613} C_VEL
LIN {X 0,Y 249.45,Z 212.41,A -85,B 0,C 180,E1 -19086.471,E2 -19086.471} C_VEL
LIN {X 0,Y 249.378,Z 212.411,A -85,B 0,C 180,E1 -19089.735,E2 -19089.735} C_VEL
LIN {X 0,Y 249.161,Z 212.444,A -85,B 0,C 180,E1 -19094.706,E2 -19094.706} C_VEL
LIN {X 0,Y 249.084,Z 212.45,A -85,B 0,C 180,E1 -19098.081,E2 -19098.081} C_VEL
LIN {X 0,Y 249.033,Z 212.468,A -85,B 0,C 180,E1 -19101.523,E2 -19101.523} C_VEL
LIN {X 0,Y 249.038,Z 212.466,A -85,B 0,C 180,E1 -19105.443,E2 -19105.443} C_VEL
LIN {X 0,Y 249.026,Z 212.467,A -85,B 0,C 180,E1 -19108.975,E2 -19108.975} C_VEL
LIN {X 0,Y 249.009,Z 212.466,A -85,B 0,C 180,E1 -19111.945,E2 -19111.945} C_VEL
LIN {X 0,Y 248.802,Z 212.807,A -85,B 0,C 180,E1 -19112.844,E2 -19112.844} C_VEL
LIN {X 0,Y 248.19,Z 213.693,A -85,B 0,C 180,E1 -19113.718,E2 -19113.718} C_VEL
LIN {X 0,Y 246.354,Z 216.411,A -85,B 0,C 180,E1 -19115.406,E2 -19115.406} C_VEL
LIN {X 0,Y 244.623,Z 219.559,A -85,B 0,C 180,E1 -19117.095,E2 -19117.095} C_VEL
LIN {X 0,Y 244.119,Z 221.73,A -85,B 0,C 180,E1 -19118.401,E2 -19118.401} C_VEL
LIN {X 0,Y 244.207,Z 222.381,A -85,B 0,C 180,E1 -19118.844,E2 -19118.844} C_VEL
LIN {X 0,Y 245.43,Z 227.759,A -85,B 0,C 180,E1 -19122.426,E2 -19122.426} C_VEL
LIN {X 0,Y 247.109,Z 235.245,A -85,B 0,C 180,E1 -19126.958,E2 -19126.958} C_VEL
LIN {X 0,Y 248.594,Z 242.06,A -85,B 0,C 180,E1 -19130.736,E2 -19130.736} C_VEL
LIN {X 0,Y 250.137,Z 249.518,A -85,B 0,C 180,E1 -19134.568,E2 -19134.568} C_VEL
LIN {X 0,Y 250.108,Z 252.102,A -85,B 0,C 180,E1 -19135.809,E2 -19135.809} C_VEL
LIN {X 0,Y 245.787,Z 265.803,A -85,B 0,C 180,E1 -19141.853,E2 -19141.853} C_VEL
LIN {X 0,Y 244.9,Z 269.2,A -85,B 0,C 180,E1 -19143.39,E2 -19143.39} C_VEL
LIN {X 0,Y 246.05,Z 281.888,A -85,B 0,C 180,E1 -19144.237,E2 -19144.237} C_VEL
LIN {X 0,Y 246.565,Z 293.488,A -85,B 0,C 180,E1 -19145.299,E2 -19145.299} C_VEL
LIN {X 0,Y 246.351,Z 305.422,A -85,B 0,C 180,E1 -19146.685,E2 -19146.685} C_VEL
LIN {X 0,Y 246.154,Z 315.629,A -85,B 0,C 180,E1 -19148.215,E2 -19148.215} C_VEL
LIN {X 0,Y 245.646,Z 324.01,A -85,B 0,C 180,E1 -19149.705,E2 -19149.705} C_VEL
LIN {X 0,Y 244.436,Z 331.021,A -85,B 0,C 180,E1 -19151.13,E2 -19151.13} C_VEL
LIN {X 0,Y 243.167,Z 339.356,A -85,B 0,C 180,E1 -19153.203,E2 -19153.203} C_VEL
LIN {X 0,Y 242.191,Z 346.348,A -85,B 0,C 180,E1 -19155.293,E2 -19155.293} C_VEL
LIN {X 0,Y 241.921,Z 349.46,A -85,B 0,C 180,E1 -19156.35,E2 -19156.35} C_VEL
LIN {X 0,Y 241.234,Z 358.523,A -85,B 0,C 180,E1 -19158.661,E2 -19158.661} C_VEL
LIN {X 0,Y 240.844,Z 366.514,A -85,B 0,C 180,E1 -19161.19,E2 -19161.19} C_VEL
LIN {X 0,Y 240.695,Z 373.04,A -85,B 0,C 180,E1 -19163.762,E2 -19163.762} C_VEL
LIN {X 0,Y 240.694,Z 378.739,A -85,B 0,C 180,E1 -19166.654,E2 -19166.654} C_VEL
LIN {X 0,Y 240.749,Z 382.392,A -85,B 0,C 180,E1 -19169.166,E2 -19169.166} C_VEL
LIN {X 0,Y 240.548,Z 384.93,A -85,B 0,C 180,E1 -19171.676,E2 -19171.676} C_VEL
LIN {X 0,Y 240.137,Z 386.801,A -85,B 0,C 180,E1 -19175.039,E2 -19175.039} C_VEL
LIN {X 0,Y 240.27,Z 387.168,A -85,B 0,C 180,E1 -19178.412,E2 -19178.412} C_VEL
LIN {X 0,Y 241.209,Z 386.102,A -85,B 0,C 180,E1 -19181.77,E2 -19181.77} C_VEL
LIN {X 0,Y 243.036,Z 383.575,A -85,B 0,C 180,E1 -19185.087,E2 -19185.087} C_VEL
LIN {X 0,Y 246.045,Z 379.64,A -85,B 0,C 180,E1 -19188.315,E2 -19188.315} C_VEL
LIN {X 0,Y 249.636,Z 374.235,A -85,B 0,C 180,E1 -19191.47,E2 -19191.47} C_VEL
LIN {X 0,Y 253.116,Z 369.12,A -85,B 0,C 180,E1 -19193.743,E2 -19193.743} C_VEL
LIN {X 0,Y 258.002,Z 361.836,A -85,B 0,C 180,E1 -19196.275,E2 -19196.275} C_VEL
LIN {X 0,Y 263.558,Z 353.063,A -85,B 0,C 180,E1 -19198.686,E2 -19198.686} C_VEL
LIN {X 0,Y 269.762,Z 342.429,A -85,B 0,C 180,E1 -19200.969,E2 -19200.969} C_VEL
LIN {X 0,Y 274.816,Z 332.061,A -85,B 0,C 180,E1 -19202.92,E2 -19202.92} C_VEL
LIN {X 0,Y 278.517,Z 322.316,A -85,B 0,C 180,E1 -19204.733,E2 -19204.733} C_VEL
LIN {X 0,Y 281.491,Z 311.874,A -85,B 0,C 180,E1 -19206.815,E2 -19206.815} C_VEL
LIN {X 0,Y 283.287,Z 303.996,A -85,B 0,C 180,E1 -19208.537,E2 -19208.537} C_VEL
LIN {X 0,Y 284.116,Z 299.847,A -85,B 0,C 180,E1 -19209.55,E2 -19209.55} C_VEL
LIN {X 0,Y 284.093,Z 298.702,A -85,B 0,C 180,E1 -19210.033,E2 -19210.033} C_VEL
LIN {X 0,Y 283.749,Z 297.065,A -85,B 0,C 180,E1 -19211.09,E2 -19211.09} C_VEL
LIN {X 0,Y 283.307,Z 296.204,A -85,B 0,C 180,E1 -19212.053,E2 -19212.053} C_VEL
LIN {X 0,Y 282.471,Z 295.298,A -85,B 0,C 180,E1 -19214.161,E2 -19214.161} C_VEL
LIN {X 0,Y 281.867,Z 295.635,A -85,B 0,C 180,E1 -19216.311,E2 -19216.311} C_VEL
LIN {X 0,Y 281.682,Z 296.337,A -85,B 0,C 180,E1 -19217.65,E2 -19217.65} C_VEL
LIN {X 0,Y 281.462,Z 298.265,A -85,B 0,C 180,E1 -19219.518,E2 -19219.518} C_VEL
LIN {X 0,Y 280.982,Z 301.509,A -85,B 0,C 180,E1 -19221.295,E2 -19221.295} C_VEL
LIN {X 0,Y 280.079,Z 308.015,A -85,B 0,C 180,E1 -19224.051,E2 -19224.051} C_VEL
LIN {X 0,Y 279.053,Z 315.353,A -85,B 0,C 180,E1 -19226.733,E2 -19226.733} C_VEL
LIN {X 0,Y 278.034,Z 320.451,A -85,B 0,C 180,E1 -19228.365,E2 -19228.365} C_VEL
LIN {X 0,Y 271.813,Z 331.487,A -85,B 0,C 180,E1 -19230.576,E2 -19230.576} C_VEL
LIN {X 0,Y 265.984,Z 340.514,A -85,B 0,C 180,E1 -19232.884,E2 -19232.884} C_VEL
LIN {X 0,Y 260.674,Z 347.914,A -85,B 0,C 180,E1 -19235.298,E2 -19235.298} C_VEL
LIN {X 0,Y 256.605,Z 353.062,A -85,B 0,C 180,E1 -19237.453,E2 -19237.453} C_VEL
LIN {X 0,Y 251.924,Z 358.388,A -85,B 0,C 180,E1 -19240.442,E2 -19240.442} C_VEL
LIN {X 0,Y 248.176,Z 362.147,A -85,B 0,C 180,E1 -19243.55,E2 -19243.55} C_VEL
LIN {X 0,Y 245.09,Z 364.423,A -85,B 0,C 180,E1 -19246.738,E2 -19246.738} C_VEL
LIN {X 0,Y 243.97,Z 365.024,A -85,B 0,C 180,E1 -19248.367,E2 -19248.367} C_VEL
LIN {X 0,Y 242.694,Z 365.307,A -85,B 0,C 180,E1 -19249.994,E2 -19249.994} C_VEL
LIN {X 0,Y 241.354,Z 364.662,A -85,B 0,C 180,E1 -19253.311,E2 -19253.311} C_VEL
LIN {X 0,Y 240.496,Z 362.577,A -85,B 0,C 180,E1 -19256.649,E2 -19256.649} C_VEL
LIN {X 0,Y 240.127,Z 359.986,A -85,B 0,C 180,E1 -19259.162,E2 -19259.162} C_VEL
LIN {X 0,Y 240.094,Z 356.463,A -85,B 0,C 180,E1 -19261.677,E2 -19261.677} C_VEL
LIN {X 0,Y 240.186,Z 351.922,A -85,B 0,C 180,E1 -19264.195,E2 -19264.195} C_VEL
LIN {X 0,Y 240.493,Z 345.153,A -85,B 0,C 180,E1 -19267.135,E2 -19267.135} C_VEL
LIN {X 0,Y 241.117,Z 336.555,A -85,B 0,C 180,E1 -19270.072,E2 -19270.072} C_VEL
LIN {X 0,Y 241.951,Z 327.345,A -85,B 0,C 180,E1 -19272.583,E2 -19272.583} C_VEL
LIN {X 0,Y 242.975,Z 317.097,A -85,B 0,C 180,E1 -19274.875,E2 -19274.875} C_VEL
LIN {X 0,Y 244.158,Z 305.703,A -85,B 0,C 180,E1 -19276.945,E2 -19276.945} C_VEL
LIN {X 0,Y 245.199,Z 294.295,A -85,B 0,C 180,E1 -19278.63,E2 -19278.63} C_VEL
LIN {X 0,Y 246.087,Z 284.028,A -85,B 0,C 180,E1 -19279.872,E2 -19279.872} C_VEL
LIN {X 0,Y 244.261,Z 271.084,A -85,B 0,C 180,E1 -19281.19,E2 -19281.19} C_VEL
LIN {X 0,Y 242.514,Z 257.18,A -85,B 0,C 180,E1 -19282.278,E2 -19282.278} C_VEL
LIN {X 0,Y 242.276,Z 254.457,A -85,B 0,C 180,E1 -19282.458,E2 -19282.458} C_VEL
LIN {X 0,Y 242.845,Z 245.923,A -85,B 0,C 180,E1 -19286.783,E2 -19286.783} C_VEL
LIN {X 0,Y 243.494,Z 237.093,A -85,B 0,C 180,E1 -19291.301,E2 -19291.301} C_VEL
LIN {X 0,Y 244.098,Z 229.595,A -85,B 0,C 180,E1 -19295.158,E2 -19295.158} C_VEL
LIN {X 0,Y 243.987,Z 224.169,A -85,B 0,C 180,E1 -19298.023,E2 -19298.023} C_VEL
LIN {X 0,Y 242.807,Z 217.43,A -85,B 0,C 180,E1 -19301.739,E2 -19301.739} C_VEL
LIN {X 0,Y 242.007,Z 213.34,A -85,B 0,C 180,E1 -19304.106,E2 -19304.106} C_VEL
LIN {X 0,Y 241.939,Z 213.347,A -85,B 0,C 180,E1 -19309.049,E2 -19309.049} C_VEL
LIN {X 0,Y 241.985,Z 213.477,A -85,B 0,C 180,E1 -19309.674,E2 -19309.674} C_VEL
LIN {X 0,Y 242.433,Z 215.632,A -85,B 0,C 180,E1 -19312.496,E2 -19312.496} C_VEL
LIN {X 0,Y 242.729,Z 217.344,A -85,B 0,C 180,E1 -19314.612,E2 -19314.612} C_VEL
LIN {X 0,Y 243.079,Z 220.755,A -85,B 0,C 180,E1 -19318.637,E2 -19318.637} C_VEL
LIN {X 0,Y 243.166,Z 222.512,A -85,B 0,C 180,E1 -19320.569,E2 -19320.569} C_VEL
LIN {X 0,Y 243.007,Z 226.13,A -85,B 0,C 180,E1 -19324.288,E2 -19324.288} C_VEL
LIN {X 0,Y 242.87,Z 230.814,A -85,B 0,C 180,E1 -19328.63,E2 -19328.63} C_VEL
LIN {X 0,Y 246.33,Z 241.395,A -85,B 0,C 180,E1 -19329.71,E2 -19329.71} C_VEL
LIN {X 0,Y 248.613,Z 250.265,A -85,B 0,C 180,E1 -19330.827,E2 -19330.827} C_VEL
LIN {X 0,Y 250.45,Z 259.802,A -85,B 0,C 180,E1 -19332.297,E2 -19332.297} C_VEL
LIN {X 0,Y 250.397,Z 262.581,A -85,B 0,C 180,E1 -19332.762,E2 -19332.762} C_VEL
LIN {X 0,Y 249.42,Z 269.854,A -85,B 0,C 180,E1 -19334.052,E2 -19334.052} C_VEL
LIN {X 0,Y 248.13,Z 277.056,A -85,B 0,C 180,E1 -19335.649,E2 -19335.649} C_VEL
LIN {X 0,Y 246.49,Z 284.064,A -85,B 0,C 180,E1 -19337.65,E2 -19337.65} C_VEL
LIN {X 0,Y 245.592,Z 288.393,A -85,B 0,C 180,E1 -19339.278,E2 -19339.278} C_VEL
LIN {X 0,Y 244.671,Z 291.899,A -85,B 0,C 180,E1 -19340.908,E2 -19340.908} C_VEL
LIN {X 0,Y 243.892,Z 295.772,A -85,B 0,C 180,E1 -19343.379,E2 -19343.379} C_VEL
LIN {X 0,Y 243.214,Z 297.606,A -85,B 0,C 180,E1 -19345.025,E2 -19345.025} C_VEL
LIN {X 0,Y 242.962,Z 298.854,A -85,B 0,C 180,E1 -19346.681,E2 -19346.681} C_VEL
LIN {X 0,Y 242.711,Z 299.617,A -85,B 0,C 180,E1 -19348.339,E2 -19348.339} C_VEL
LIN {X 0,Y 242.612,Z 299.888,A -85,B 0,C 180,E1 -19349.998,E2 -19349.998} C_VEL
LIN {X 0,Y 242.709,Z 299.652,A -85,B 0,C 180,E1 -19351.657,E2 -19351.657} C_VEL
LIN {X 0,Y 242.959,Z 298.937,A -85,B 0,C 180,E1 -19353.314,E2 -19353.314} C_VEL
LIN {X 0,Y 243.212,Z 297.738,A -85,B 0,C 180,E1 -19354.971,E2 -19354.971} C_VEL
LIN {X 0,Y 244.216,Z 294.818,A -85,B 0,C 180,E1 -19357.438,E2 -19357.438} C_VEL
LIN {X 0,Y 244.911,Z 290.543,A -85,B 0,C 180,E1 -19359.912,E2 -19359.912} C_VEL
LIN {X 0,Y 245.613,Z 288.695,A -85,B 0,C 180,E1 -19360.717,E2 -19360.717} C_VEL
LIN {X 0,Y 246.453,Z 284.446,A -85,B 0,C 180,E1 -19362.347,E2 -19362.347} C_VEL
LIN {X 0,Y 248.107,Z 277.593,A -85,B 0,C 180,E1 -19364.348,E2 -19364.348} C_VEL
LIN {X 0,Y 249.354,Z 270.512,A -85,B 0,C 180,E1 -19365.948,E2 -19365.948} C_VEL
LIN {X 0,Y 250.231,Z 263.908,A -85,B 0,C 180,E1 -19367.157,E2 -19367.157} C_VEL
LIN {X 0,Y 250.484,Z 260.018,A -85,B 0,C 180,E1 -19367.8,E2 -19367.8} C_VEL
LIN {X 0,Y 248.781,Z 250.761,A -85,B 0,C 180,E1 -19369.23,E2 -19369.23} C_VEL
LIN {X 0,Y 246.467,Z 241.821,A -85,B 0,C 180,E1 -19370.376,E2 -19370.376} C_VEL
LIN {X 0,Y 242.856,Z 230.577,A -85,B 0,C 180,E1 -19371.57,E2 -19371.57} C_VEL
LIN {X 0,Y 243.06,Z 225.677,A -85,B 0,C 180,E1 -19376.316,E2 -19376.316} C_VEL
LIN {X 0,Y 243.144,Z 222.277,A -85,B 0,C 180,E1 -19379.871,E2 -19379.871} C_VEL
LIN {X 0,Y 242.959,Z 219.212,A -85,B 0,C 180,E1 -19383.337,E2 -19383.337} C_VEL
LIN {X 0,Y 242.449,Z 215.79,A -85,B 0,C 180,E1 -19387.495,E2 -19387.495} C_VEL
LIN {X 0,Y 241.943,Z 213.348,A -85,B 0,C 180,E1 -19390.952,E2 -19390.952} C_VEL
LIN {X 0,Y 241.93,Z 213.346,A -85,B 0,C 180,E1 -19394.199,E2 -19394.199} C_VEL
LIN {X 0,Y 241.945,Z 213.349,A -85,B 0,C 180,E1 -19398.079,E2 -19398.079} C_VEL
LIN {X 0,Y 241.987,Z 213.335,A -85,B 0,C 180,E1 -19402.417,E2 -19402.417} C_VEL
LIN {X 0,Y 241.98,Z 213.334,A -85,B 0,C 180,E1 -19406.507,E2 -19406.507} C_VEL
LIN {X 0,Y 242.029,Z 213.326,A -85,B 0,C 180,E1 -19410.586,E2 -19410.586} C_VEL
LIN {X 0,Y 242.059,Z 213.323,A -85,B 0,C 180,E1 -19414.182,E2 -19414.182} C_VEL
LIN {X 0,Y 242.044,Z 213.33,A -85,B 0,C 180,E1 -19418.296,E2 -19418.296} C_VEL
LIN {X 0,Y 242.154,Z 213.316,A -85,B 0,C 180,E1 -19423.277,E2 -19423.277} C_VEL
LIN {X 0,Y 242.171,Z 213.316,A -85,B 0,C 180,E1 -19428.279,E2 -19428.279} C_VEL
LIN {X 0,Y 242.39,Z 213.286,A -85,B 0,C 180,E1 -19431.664,E2 -19431.664} C_VEL
LIN {X 0,Y 242.246,Z 213.294,A -85,B 0,C 180,E1 -19435.007,E2 -19435.007} C_VEL
LIN {X 0,Y 242.626,Z 213.26,A -85,B 0,C 180,E1 -19438.34,E2 -19438.34} C_VEL
LIN {X 0,Y 242.625,Z 213.259,A -85,B 0,C 180,E1 -19441.66,E2 -19441.66} C_VEL
LIN {X 0,Y 242.422,Z 213.287,A -85,B 0,C 180,E1 -19446.659,E2 -19446.659} C_VEL
LIN {X 0,Y 242.304,Z 213.293,A -85,B 0,C 180,E1 -19450.022,E2 -19450.022} C_VEL
LIN {X 0,Y 242.116,Z 213.327,A -85,B 0,C 180,E1 -19455.144,E2 -19455.144} C_VEL
LIN {X 0,Y 242.021,Z 213.334,A -85,B 0,C 180,E1 -19458.628,E2 -19458.628} C_VEL
LIN {X 0,Y 241.963,Z 213.346,A -85,B 0,C 180,E1 -19462.185,E2 -19462.185} C_VEL
LIN {X 0,Y 241.977,Z 213.345,A -85,B 0,C 180,E1 -19465.827,E2 -19465.827} C_VEL
LIN {X 0,Y 241.959,Z 213.347,A -85,B 0,C 180,E1 -19469.59,E2 -19469.59} C_VEL
LIN {X 0,Y 241.996,Z 213.501,A -85,B 0,C 180,E1 -19471.95,E2 -19471.95} C_VEL
LIN {X 0,Y 243.293,Z 218.448,A -85,B 0,C 180,E1 -19476.022,E2 -19476.022} C_VEL
LIN {X 0,Y 244.207,Z 222.381,A -85,B 0,C 180,E1 -19478.844,E2 -19478.844} C_VEL
LIN {X 0,Y 244.047,Z 224.478,A -85,B 0,C 180,E1 -19480.137,E2 -19480.137} C_VEL
LIN {X 0,Y 242.034,Z 228.561,A -85,B 0,C 180,E1 -19482.213,E2 -19482.213} C_VEL
LIN {X 0,Y 240.274,Z 231.965,A -85,B 0,C 180,E1 -19483.889,E2 -19483.889} C_VEL
LIN {X 0,Y 239.73,Z 234.374,A -85,B 0,C 180,E1 -19485.188,E2 -19485.188} C_VEL
LIN {X 0,Y 239.811,Z 235.12,A -85,B 0,C 180,E1 -19485.629,E2 -19485.629} C_VEL
LIN {X 0,Y 241.195,Z 241.233,A -85,B 0,C 180,E1 -19489.253,E2 -19489.253} C_VEL
LIN {X 0,Y 243.012,Z 250.116,A -85,B 0,C 180,E1 -19494.074,E2 -19494.074} C_VEL
LIN {X 0,Y 243.221,Z 252.356,A -85,B 0,C 180,E1 -19495.205,E2 -19495.205} C_VEL
LIN {X 0,Y 241.58,Z 257.454,A -85,B 0,C 180,E1 -19497.529,E2 -19497.529} C_VEL
LIN {X 0,Y 238.18,Z 268.571,A -85,B 0,C 180,E1 -19502.669,E2 -19502.669} C_VEL
LIN {X 0,Y 239.291,Z 281.051,A -85,B 0,C 180,E1 -19503.531,E2 -19503.531} C_VEL
LIN {X 0,Y 239.845,Z 293.258,A -85,B 0,C 180,E1 -19504.694,E2 -19504.694} C_VEL
LIN {X 0,Y 239.605,Z 304.112,A -85,B 0,C 180,E1 -19505.988,E2 -19505.988} C_VEL
LIN {X 0,Y 239.307,Z 314.422,A -85,B 0,C 180,E1 -19507.558,E2 -19507.558} C_VEL
LIN {X 0,Y 238.873,Z 322.883,A -85,B 0,C 180,E1 -19509.103,E2 -19509.103} C_VEL
LIN {X 0,Y 237.335,Z 331.694,A -85,B 0,C 180,E1 -19510.992,E2 -19510.992} C_VEL
LIN {X 0,Y 236.284,Z 338.301,A -85,B 0,C 180,E1 -19512.699,E2 -19512.699} C_VEL
LIN {X 0,Y 235.231,Z 345.311,A -85,B 0,C 180,E1 -19514.848,E2 -19514.848} C_VEL
LIN {X 0,Y 234.671,Z 350.915,A -85,B 0,C 180,E1 -19516.912,E2 -19516.912} C_VEL
LIN {X 0,Y 233.988,Z 360.614,A -85,B 0,C 180,E1 -19519.62,E2 -19519.62} C_VEL
LIN {X 0,Y 233.773,Z 368.352,A -85,B 0,C 180,E1 -19522.314,E2 -19522.314} C_VEL
LIN {X 0,Y 233.694,Z 374.084,A -85,B 0,C 180,E1 -19524.826,E2 -19524.826} C_VEL
LIN {X 0,Y 233.74,Z 378.743,A -85,B 0,C 180,E1 -19527.417,E2 -19527.417} C_VEL
LIN {X 0,Y 233.75,Z 382.22,A -85,B 0,C 180,E1 -19530.002,E2 -19530.002} C_VEL
LIN {X 0,Y 233.521,Z 383.908,A -85,B 0,C 180,E1 -19531.727,E2 -19531.727} C_VEL
LIN {X 0,Y 233.068,Z 386.047,A -85,B 0,C 180,E1 -19535.192,E2 -19535.192} C_VEL
LIN {X 0,Y 233.225,Z 386.668,A -85,B 0,C 180,E1 -19538.668,E2 -19538.668} C_VEL
LIN {X 0,Y 234.247,Z 385.853,A -85,B 0,C 180,E1 -19542.126,E2 -19542.126} C_VEL
LIN {X 0,Y 236.197,Z 383.667,A -85,B 0,C 180,E1 -19545.535,E2 -19545.535} C_VEL
LIN {X 0,Y 239.323,Z 380.064,A -85,B 0,C 180,E1 -19548.848,E2 -19548.848} C_VEL
LIN {X 0,Y 243.085,Z 375.041,A -85,B 0,C 180,E1 -19552.079,E2 -19552.079} C_VEL
LIN {X 0,Y 246.729,Z 370.252,A -85,B 0,C 180,E1 -19554.397,E2 -19554.397} C_VEL
LIN {X 0,Y 251.796,Z 363.455,A -85,B 0,C 180,E1 -19556.974,E2 -19556.974} C_VEL
LIN {X 0,Y 257.536,Z 355.229,A -85,B 0,C 180,E1 -19559.422,E2 -19559.422} C_VEL
LIN {X 0,Y 263.967,Z 345.291,A -85,B 0,C 180,E1 -19561.726,E2 -19561.726} C_VEL
LIN {X 0,Y 269.387,Z 335.555,A -85,B 0,C 180,E1 -19563.671,E2 -19563.671} C_VEL
LIN {X 0,Y 273.294,Z 326.899,A -85,B 0,C 180,E1 -19565.355,E2 -19565.355} C_VEL
LIN {X 0,Y 276.638,Z 317.709,A -85,B 0,C 180,E1 -19567.249,E2 -19567.249} C_VEL
LIN {X 0,Y 279.08,Z 309.744,A -85,B 0,C 180,E1 -19569.02,E2 -19569.02} C_VEL
LIN {X 0,Y 280.36,Z 305.074,A -85,B 0,C 180,E1 -19570.188,E2 -19570.188} C_VEL
LIN {X 0,Y 280.246,Z 303.292,A -85,B 0,C 180,E1 -19571.206,E2 -19571.206} C_VEL
LIN {X 0,Y 279.441,Z 301.908,A -85,B 0,C 180,E1 -19573.167,E2 -19573.167} C_VEL
LIN {X 0,Y 278.766,Z 301.635,A -85,B 0,C 180,E1 -19575.097,E2 -19575.097} C_VEL
LIN {X 0,Y 278.3,Z 302.274,A -85,B 0,C 180,E1 -19577.086,E2 -19577.086} C_VEL
LIN {X 0,Y 277.765,Z 304.44,A -85,B 0,C 180,E1 -19579.384,E2 -19579.384} C_VEL
LIN {X 0,Y 276.926,Z 307.709,A -85,B 0,C 180,E1 -19581.16,E2 -19581.16} C_VEL
LIN {X 0,Y 275.445,Z 314.376,A -85,B 0,C 180,E1 -19584.066,E2 -19584.066} C_VEL
LIN {X 0,Y 274.031,Z 320.724,A -85,B 0,C 180,E1 -19586.479,E2 -19586.479} C_VEL
LIN {X 0,Y 273.339,Z 323.153,A -85,B 0,C 180,E1 -19587.32,E2 -19587.32} C_VEL
LIN {X 0,Y 272.714,Z 324.568,A -85,B 0,C 180,E1 -19587.674,E2 -19587.674} C_VEL
LIN {X 0,Y 266.084,Z 334.931,A -85,B 0,C 180,E1 -19589.878,E2 -19589.878} C_VEL
LIN {X 0,Y 260.07,Z 343.358,A -85,B 0,C 180,E1 -19592.215,E2 -19592.215} C_VEL
LIN {X 0,Y 254.538,Z 350.244,A -85,B 0,C 180,E1 -19594.661,E2 -19594.661} C_VEL
LIN {X 0,Y 250.314,Z 355.025,A -85,B 0,C 180,E1 -19596.854,E2 -19596.854} C_VEL
LIN {X 0,Y 246.58,Z 358.86,A -85,B 0,C 180,E1 -19599.128,E2 -19599.128} C_VEL
LIN {X 0,Y 243.324,Z 361.821,A -85,B 0,C 180,E1 -19601.475,E2 -19601.475} C_VEL
LIN {X 0,Y 239.722,Z 364.497,A -85,B 0,C 180,E1 -19604.701,E2 -19604.701} C_VEL
LIN {X 0,Y 237.053,Z 365.724,A -85,B 0,C 180,E1 -19608.022,E2 -19608.022} C_VEL
LIN {X 0,Y 235.733,Z 365.823,A -85,B 0,C 180,E1 -19609.695,E2 -19609.695} C_VEL
LIN {X 0,Y 234.312,Z 364.918,A -85,B 0,C 180,E1 -19613.109,E2 -19613.109} C_VEL
LIN {X 0,Y 233.841,Z 363.923,A -85,B 0,C 180,E1 -19614.827,E2 -19614.827} C_VEL
LIN {X 0,Y 233.154,Z 360.76,A -85,B 0,C 180,E1 -19618.273,E2 -19618.273} C_VEL
LIN {X 0,Y 232.989,Z 357.344,A -85,B 0,C 180,E1 -19620.864,E2 -19620.864} C_VEL
LIN {X 0,Y 233.097,Z 352.934,A -85,B 0,C 180,E1 -19623.457,E2 -19623.457} C_VEL
LIN {X 0,Y 233.276,Z 346.36,A -85,B 0,C 180,E1 -19626.487,E2 -19626.487} C_VEL
LIN {X 0,Y 233.765,Z 339.297,A -85,B 0,C 180,E1 -19629.082,E2 -19629.082} C_VEL
LIN {X 0,Y 234.509,Z 330.646,A -85,B 0,C 180,E1 -19631.671,E2 -19631.671} C_VEL
LIN {X 0,Y 235.299,Z 321.989,A -85,B 0,C 180,E1 -19633.825,E2 -19633.825} C_VEL
LIN {X 0,Y 236.424,Z 311.632,A -85,B 0,C 180,E1 -19635.96,E2 -19635.96} C_VEL
LIN {X 0,Y 237.545,Z 300.276,A -85,B 0,C 180,E1 -19637.876,E2 -19637.876} C_VEL
LIN {X 0,Y 238.782,Z 287.311,A -85,B 0,C 180,E1 -19639.631,E2 -19639.631} C_VEL
LIN {X 0,Y 238.897,Z 283.063,A -85,B 0,C 180,E1 -19640.127,E2 -19640.127} C_VEL
LIN {X 0,Y 236.762,Z 268.506,A -85,B 0,C 180,E1 -19641.606,E2 -19641.606} C_VEL
LIN {X 0,Y 235.255,Z 254.79,A -85,B 0,C 180,E1 -19642.656,E2 -19642.656} C_VEL
LIN {X 0,Y 235.865,Z 245.391,A -85,B 0,C 180,E1 -19647.506,E2 -19647.506} C_VEL
LIN {X 0,Y 236.603,Z 236.146,A -85,B 0,C 180,E1 -19652.322,E2 -19652.322} C_VEL
LIN {X 0,Y 237.08,Z 230.446,A -85,B 0,C 180,E1 -19655.314,E2 -19655.314} C_VEL
LIN {X 0,Y 237.07,Z 226.186,A -85,B 0,C 180,E1 -19657.598,E2 -19657.598} C_VEL
LIN {X 0,Y 236.115,Z 220.224,A -85,B 0,C 180,E1 -19660.907,E2 -19660.907} C_VEL
LIN {X 0,Y 234.952,Z 214.217,A -85,B 0,C 180,E1 -19664.362,E2 -19664.362} C_VEL
LIN {X 0,Y 234.915,Z 214.307,A -85,B 0,C 180,E1 -19668.412,E2 -19668.412} C_VEL
LIN {X 0,Y 235.349,Z 216.333,A -85,B 0,C 180,E1 -19671.161,E2 -19671.161} C_VEL
LIN {X 0,Y 235.877,Z 219.731,A -85,B 0,C 180,E1 -19675.518,E2 -19675.518} C_VEL
LIN {X 0,Y 236.098,Z 221.462,A -85,B 0,C 180,E1 -19677.599,E2 -19677.599} C_VEL
LIN {X 0,Y 236.191,Z 223.259,A -85,B 0,C 180,E1 -19679.646,E2 -19679.646} C_VEL
LIN {X 0,Y 236.12,Z 226.84,A -85,B 0,C 180,E1 -19683.481,E2 -19683.481} C_VEL
LIN {X 0,Y 235.924,Z 231.453,A -85,B 0,C 180,E1 -19687.873,E2 -19687.873} C_VEL
LIN {X 0,Y 239.541,Z 242.387,A -85,B 0,C 180,E1 -19689.047,E2 -19689.047} C_VEL
LIN {X 0,Y 241.937,Z 251.55,A -85,B 0,C 180,E1 -19690.266,E2 -19690.266} C_VEL
LIN {X 0,Y 243.869,Z 262.088,A -85,B 0,C 180,E1 -19691.994,E2 -19691.994} C_VEL
LIN {X 0,Y 242.859,Z 269.938,A -85,B 0,C 180,E1 -19693.393,E2 -19693.393} C_VEL
LIN {X 0,Y 241.697,Z 276.438,A -85,B 0,C 180,E1 -19694.827,E2 -19694.827} C_VEL
LIN {X 0,Y 240.301,Z 282.526,A -85,B 0,C 180,E1 -19696.467,E2 -19696.467} C_VEL
LIN {X 0,Y 239.073,Z 287.356,A -85,B 0,C 180,E1 -19698.123,E2 -19698.123} C_VEL
LIN {X 0,Y 238.029,Z 291.255,A -85,B 0,C 180,E1 -19699.794,E2 -19699.794} C_VEL
LIN {X 0,Y 237.261,Z 295.611,A -85,B 0,C 180,E1 -19702.338,E2 -19702.338} C_VEL
LIN {X 0,Y 236.214,Z 298.583,A -85,B 0,C 180,E1 -19704.877,E2 -19704.877} C_VEL
LIN {X 0,Y 235.947,Z 299.829,A -85,B 0,C 180,E1 -19706.583,E2 -19706.583} C_VEL
LIN {X 0,Y 235.686,Z 300.591,A -85,B 0,C 180,E1 -19708.289,E2 -19708.289} C_VEL
LIN {X 0,Y 235.585,Z 300.862,A -85,B 0,C 180,E1 -19709.998,E2 -19709.998} C_VEL
LIN {X 0,Y 235.685,Z 300.625,A -85,B 0,C 180,E1 -19711.707,E2 -19711.707} C_VEL
LIN {X 0,Y 235.944,Z 299.91,A -85,B 0,C 180,E1 -19713.413,E2 -19713.413} C_VEL
LIN {X 0,Y 236.212,Z 298.713,A -85,B 0,C 180,E1 -19715.119,E2 -19715.119} C_VEL
LIN {X 0,Y 237.249,Z 295.793,A -85,B 0,C 180,E1 -19717.658,E2 -19717.658} C_VEL
LIN {X 0,Y 237.988,Z 291.529,A -85,B 0,C 180,E1 -19720.204,E2 -19720.204} C_VEL
LIN {X 0,Y 238.706,Z 289.686,A -85,B 0,C 180,E1 -19721.031,E2 -19721.031} C_VEL
LIN {X 0,Y 239.593,Z 285.452,A -85,B 0,C 180,E1 -19722.707,E2 -19722.707} C_VEL
LIN {X 0,Y 241.315,Z 278.643,A -85,B 0,C 180,E1 -19724.761,E2 -19724.761} C_VEL
LIN {X 0,Y 242.626,Z 271.604,A -85,B 0,C 180,E1 -19726.402,E2 -19726.402} C_VEL
LIN {X 0,Y 243.606,Z 264.586,A -85,B 0,C 180,E1 -19727.722,E2 -19727.722} C_VEL
LIN {X 0,Y 243.743,Z 261.175,A -85,B 0,C 180,E1 -19728.316,E2 -19728.316} C_VEL
LIN {X 0,Y 242.092,Z 252.066,A -85,B 0,C 180,E1 -19729.79,E2 -19729.79} C_VEL
LIN {X 0,Y 239.731,Z 242.83,A -85,B 0,C 180,E1 -19731.032,E2 -19731.032} C_VEL
LIN {X 0,Y 235.9,Z 231.28,A -85,B 0,C 180,E1 -19732.289,E2 -19732.289} C_VEL
LIN {X 0,Y 236.106,Z 226.79,A -85,B 0,C 180,E1 -19736.748,E2 -19736.748} C_VEL
LIN {X 0,Y 236.181,Z 223.411,A -85,B 0,C 180,E1 -19740.386,E2 -19740.386} C_VEL
LIN {X 0,Y 236.04,Z 220.693,A -85,B 0,C 180,E1 -19743.52,E2 -19743.52} C_VEL
LIN {X 0,Y 235.669,Z 218.165,A -85,B 0,C 180,E1 -19746.611,E2 -19746.611} C_VEL
LIN {X 0,Y 235.331,Z 216.307,A -85,B 0,C 180,E1 -19749.061,E2 -19749.061} C_VEL
LIN {X 0,Y 234.892,Z 214.224,A -85,B 0,C 180,E1 -19751.945,E2 -19751.945} C_VEL
LIN {X 0,Y 234.916,Z 214.218,A -85,B 0,C 180,E1 -19756.52,E2 -19756.52} C_VEL
LIN {X 0,Y 234.948,Z 214.22,A -85,B 0,C 180,E1 -19761.084,E2 -19761.084} C_VEL
LIN {X 0,Y 234.943,Z 214.215,A -85,B 0,C 180,E1 -19765.364,E2 -19765.364} C_VEL
LIN {X 0,Y 234.924,Z 214.216,A -85,B 0,C 180,E1 -19769.431,E2 -19769.431} C_VEL
LIN {X 0,Y 234.986,Z 214.207,A -85,B 0,C 180,E1 -19773.792,E2 -19773.792} C_VEL
LIN {X 0,Y 235.002,Z 214.201,A -85,B 0,C 180,E1 -19778.969,E2 -19778.969} C_VEL
LIN {X 0,Y 235.087,Z 214.199,A -85,B 0,C 180,E1 -19783.058,E2 -19783.058} C_VEL
LIN {X 0,Y 235.105,Z 214.198,A -85,B 0,C 180,E1 -19787.921,E2 -19787.921} C_VEL
LIN {X 0,Y 235.321,Z 214.163,A -85,B 0,C 180,E1 -19791.412,E2 -19791.412} C_VEL
LIN {X 0,Y 235.382,Z 214.162,A -85,B 0,C 180,E1 -19793.141,E2 -19793.141} C_VEL
LIN {X 0,Y 235.585,Z 214.137,A -85,B 0,C 180,E1 -19798.29,E2 -19798.29} C_VEL
LIN {X 0,Y 235.584,Z 214.136,A -85,B 0,C 180,E1 -19801.709,E2 -19801.709} C_VEL
LIN {X 0,Y 235.393,Z 214.164,A -85,B 0,C 180,E1 -19806.859,E2 -19806.859} C_VEL
LIN {X 0,Y 235.227,Z 214.177,A -85,B 0,C 180,E1 -19810.327,E2 -19810.327} C_VEL
LIN {X 0,Y 235.064,Z 214.206,A -85,B 0,C 180,E1 -19815.61,E2 -19815.61} C_VEL
LIN {X 0,Y 234.959,Z 214.22,A -85,B 0,C 180,E1 -19819.21,E2 -19819.21} C_VEL
LIN {X 0,Y 234.899,Z 214.227,A -85,B 0,C 180,E1 -19822.889,E2 -19822.889} C_VEL
LIN {X 0,Y 234.916,Z 214.227,A -85,B 0,C 180,E1 -19826.664,E2 -19826.664} C_VEL
LIN {X 0,Y 234.903,Z 214.326,A -85,B 0,C 180,E1 -19830.343,E2 -19830.343} C_VEL
LIN {X 0,Y 236.117,Z 218.936,A -85,B 0,C 180,E1 -19834.439,E2 -19834.439} C_VEL
LIN {X 0,Y 237.482,Z 224.638,A -85,B 0,C 180,E1 -19838.778,E2 -19838.778} C_VEL
LIN {X 0,Y 238.764,Z 230.285,A -85,B 0,C 180,E1 -19842.623,E2 -19842.623} C_VEL
LIN {X 0,Y 239.811,Z 235.12,A -85,B 0,C 180,E1 -19845.629,E2 -19845.629} C_VEL
LIN {X 0,Y 239.64,Z 237.455,A -85,B 0,C 180,E1 -19846.924,E2 -19846.924} C_VEL
LIN {X 0,Y 237.623,Z 241.769,A -85,B 0,C 180,E1 -19849.014,E2 -19849.014} C_VEL
LIN {X 0,Y 235.886,Z 245.324,A -85,B 0,C 180,E1 -19850.703,E2 -19850.703} C_VEL
LIN {X 0,Y 235.376,Z 247.895,A -85,B 0,C 180,E1 -19852.008,E2 -19852.008} C_VEL
LIN {X 0,Y 235.471,Z 248.71,A -85,B 0,C 180,E1 -19852.45,E2 -19852.45} C_VEL
LIN {X 0,Y 236.297,Z 252.72,A -85,B 0,C 180,E1 -19854.614,E2 -19854.614} C_VEL
LIN {X 0,Y 235.982,Z 254.592,A -85,B 0,C 180,E1 -19855.541,E2 -19855.541} C_VEL
LIN {X 0,Y 231.488,Z 267.914,A -85,B 0,C 180,E1 -19861.902,E2 -19861.902} C_VEL
LIN {X 0,Y 232.647,Z 280.671,A -85,B 0,C 180,E1 -19862.83,E2 -19862.83} C_VEL
LIN {X 0,Y 233.115,Z 293.325,A -85,B 0,C 180,E1 -19864.082,E2 -19864.082} C_VEL
LIN {X 0,Y 232.805,Z 304.399,A -85,B 0,C 180,E1 -19865.478,E2 -19865.478} C_VEL
LIN {X 0,Y 232.403,Z 314.471,A -85,B 0,C 180,E1 -19867.089,E2 -19867.089} C_VEL
LIN {X 0,Y 231.961,Z 322.799,A -85,B 0,C 180,E1 -19868.683,E2 -19868.683} C_VEL
LIN {X 0,Y 230.576,Z 330.618,A -85,B 0,C 180,E1 -19870.413,E2 -19870.413} C_VEL
LIN {X 0,Y 229.404,Z 337.245,A -85,B 0,C 180,E1 -19872.163,E2 -19872.163} C_VEL
LIN {X 0,Y 228.282,Z 344.271,A -85,B 0,C 180,E1 -19874.375,E2 -19874.375} C_VEL
LIN {X 0,Y 227.547,Z 351.014,A -85,B 0,C 180,E1 -19877.063,E2 -19877.063} C_VEL
LIN {X 0,Y 227.465,Z 352.154,A -85,B 0,C 180,E1 -19877.512,E2 -19877.512} C_VEL
LIN {X 0,Y 226.902,Z 361.18,A -85,B 0,C 180,E1 -19880.194,E2 -19880.194} C_VEL
LIN {X 0,Y 226.753,Z 368.439,A -85,B 0,C 180,E1 -19882.881,E2 -19882.881} C_VEL
LIN {X 0,Y 226.705,Z 374.189,A -85,B 0,C 180,E1 -19885.557,E2 -19885.557} C_VEL
LIN {X 0,Y 226.763,Z 378.678,A -85,B 0,C 180,E1 -19888.226,E2 -19888.226} C_VEL
LIN {X 0,Y 226.746,Z 381.009,A -85,B 0,C 180,E1 -19890.002,E2 -19890.002} C_VEL
LIN {X 0,Y 226.493,Z 382.848,A -85,B 0,C 180,E1 -19891.78,E2 -19891.78} C_VEL
LIN {X 0,Y 226.014,Z 385.198,A -85,B 0,C 180,E1 -19895.355,E2 -19895.355} C_VEL
LIN {X 0,Y 226.202,Z 386.094,A -85,B 0,C 180,E1 -19898.939,E2 -19898.939} C_VEL
LIN {X 0,Y 227.279,Z 385.599,A -85,B 0,C 180,E1 -19902.503,E2 -19902.503} C_VEL
LIN {X 0,Y 229.349,Z 383.693,A -85,B 0,C 180,E1 -19906.011,E2 -19906.011} C_VEL
LIN {X 0,Y 232.611,Z 380.436,A -85,B 0,C 180,E1 -19909.414,E2 -19909.414} C_VEL
LIN {X 0,Y 236.562,Z 375.838,A -85,B 0,C 180,E1 -19912.721,E2 -19912.721} C_VEL
LIN {X 0,Y 240.357,Z 371.376,A -85,B 0,C 180,E1 -19915.088,E2 -19915.088} C_VEL
LIN {X 0,Y 245.616,Z 365.038,A -85,B 0,C 180,E1 -19917.711,E2 -19917.711} C_VEL
LIN {X 0,Y 252.484,Z 356.091,A -85,B 0,C 180,E1 -19920.533,E2 -19920.533} C_VEL
LIN {X 0,Y 259.195,Z 346.594,A -85,B 0,C 180,E1 -19922.842,E2 -19922.842} C_VEL
LIN {X 0,Y 265.761,Z 335.675,A -85,B 0,C 180,E1 -19925.114,E2 -19925.114} C_VEL
LIN {X 0,Y 270.382,Z 326.137,A -85,B 0,C 180,E1 -19927.101,E2 -19927.101} C_VEL
LIN {X 0,Y 273.737,Z 317.705,A -85,B 0,C 180,E1 -19928.997,E2 -19928.997} C_VEL
LIN {X 0,Y 276.484,Z 310.17,A -85,B 0,C 180,E1 -19930.87,E2 -19930.87} C_VEL
LIN {X 0,Y 276.493,Z 309.314,A -85,B 0,C 180,E1 -19931.369,E2 -19931.369} C_VEL
LIN {X 0,Y 275.689,Z 307.938,A -85,B 0,C 180,E1 -19933.498,E2 -19933.498} C_VEL
LIN {X 0,Y 274.912,Z 307.917,A -85,B 0,C 180,E1 -19935.711,E2 -19935.711} C_VEL
LIN {X 0,Y 274.167,Z 309.321,A -85,B 0,C 180,E1 -19938.204,E2 -19938.204} C_VEL
LIN {X 0,Y 273.979,Z 309.936,A -85,B 0,C 180,E1 -19938.842,E2 -19938.842} C_VEL
LIN {X 0,Y 272.93,Z 312.881,A -85,B 0,C 180,E1 -19940.582,E2 -19940.582} C_VEL
LIN {X 0,Y 270.897,Z 319.24,A -85,B 0,C 180,E1 -19943.54,E2 -19943.54} C_VEL
LIN {X 0,Y 269.003,Z 325.338,A -85,B 0,C 180,E1 -19946.005,E2 -19946.005} C_VEL
LIN {X 0,Y 268.262,Z 327.135,A -85,B 0,C 180,E1 -19946.622,E2 -19946.622} C_VEL
LIN {X 0,Y 261.364,Z 337.057,A -85,B 0,C 180,E1 -19948.827,E2 -19948.827} C_VEL
LIN {X 0,Y 255.051,Z 345.114,A -85,B 0,C 180,E1 -19951.17,E2 -19951.17} C_VEL
LIN {X 0,Y 249.991,Z 350.874,A -85,B 0,C 180,E1 -19953.269,E2 -19953.269} C_VEL
LIN {X 0,Y 245.419,Z 355.611,A -85,B 0,C 180,E1 -19955.466,E2 -19955.466} C_VEL
